// TwinCAT 3 PLC project PLC
// ProgramVersion: 3.1.4022.1
// CompilerDefines: VISU_USEWSTRING
// libraries:
//   Tc2_Drive, * (Beckhoff Automation GmbH)
//   Tc2_EtherCAT, * (Beckhoff Automation GmbH)
//   Tc2_MC2, * (Beckhoff Automation GmbH)
//   Tc2_MC2_Drive, * (Beckhoff Automation GmbH)
//   Tc2_NCI, * (Beckhoff Automation GmbH)
//   Tc2_NcKinematicTransformation, * (Beckhoff Automation GmbH)
//   Tc2_Standard, * (Beckhoff Automation GmbH)
//   Tc2_System, * (Beckhoff Automation GmbH)
//   Tc2_Utilities, * (Beckhoff Automation GmbH)
//   Tc3_McCoordinatedMotion, * (Beckhoff Automation GmbH)
//   Tc3_Module, * (Beckhoff Automation GmbH)
//   VisuDialogs, * (System)
//   VisuElemEventTable,1.0.2.0,System
//   VisuSymbols,newest,System
// project tree:
//   DUTs/ uBYTE_BOOL_MX2.TcDUT, uWORD_BOOL_MX2.TcDUT, E_ColumState.TcDUT, E_LineMachineCommand.TcDUT, E_LineMachineMode.TcDUT, E_MachineCommand.TcDUT, E_MachineMode.TcDUT, E_MachineState.TcDUT, ST_AX5000Diag.TcDUT, ST_ChannelSignals.TcDUT
//   DUTs/E_CaseCloser/ E_CaseCloserMachineState.TcDUT
//   DUTs/E_CaseErector/ E_CaseErectorMachineState.TcDUT
//   DUTs/E_Gantry/ E_GantryMachineState.TcDUT
//   DUTs/HMI/ ST_MachineMode.TcDUT, ST_ManualMode.TcDUT
//   DUTs/NCI/ E_NCIOpModes.TcDUT, ST_NCIChannelState.TcDUT
//   GVLs/ Global_HMI.TcGVL, GVL.TcGVL, GVL_AXIS.TcGVL, GVL_EventsSimple.TcGVL, GVL_GLOBAL.TcGVL, GVL_HMI.TcGVL, GVL_IO.TcGVL, GVL_IO_K.TcGVL, GVL_IO_P.TcGVL, GVL_Kolumna.TcGVL, GVL_Machine.TcGVL, GVL_MachineMaintenance.TcGVL, GVL_NCI.TcGVL, GVL_Omron.TcGVL, GVL_Recipe.TcGVL, GVL_RecipeTable.TcGVL, GVL_SafetyFrom_RT2.TcGVL, GVL_Zak_IO.TcGVL
//   / PlcTask.TcTTO, Recepty.TcTTO, VISU_TASK.TcTTO
//   POUs/Eventy/ FB_SimpleEventLog.TcPOU, P_EventsSimple.TcPOU
//   POUs/FB/ FB_AxisDiag.TcPOU, FB_Button.TcPOU, FB_INV000_MX2_Alarm.TcPOU, FB_INV003_MX2_ECT.TcPOU, FB_Kierownica.TcPOU, FB_K_Auto.TcPOU, FB_Licznik.TcPOU, FB_Magazyn.TcPOU, FB_MX2.TcPOU, FB_MX2_POS.TcPOU, FB_Prawidlo.TcPOU, F_4BYTES_TO_DWORD.TcPOU
//   POUs/Programy/Hbot/AxisOnline/DUTsAxisOnline/FBsIO/ ST_FBCoESetPositionOffsetIO.TcDUT, ST_FBGetDriveRefIO.TcDUT, ST_FBHoldingBrakeCtrlIO.TcDUT, ST_FBMotorMonitoringIO.TcDUT, ST_FBNcSWLimitSwitchCtrlIO.TcDUT, ST_FBReadChannelErrorCodeIO.TcDUT, ST_FBSetPositionOffsetIO.TcDUT, ST_McAxisOnlineErrorCollection.TcDUT, ST_McAxisStatus.TcDUT, ST_MCHaltIO.TcDUT, ST_MCHomeIO.TcDUT, ST_MCJogIO.TcDUT, ST_MCMoveAbsoluteIO.TcDUT, ST_MCMoveModuloIO.TcDUT, ST_MCMoveRelativeIO.TcDUT, ST_MCMoveVelocityIO.TcDUT, ST_MCPowerIO.TcDUT, ST_MCReadDriveAddressIO.TcDUT, ST_MCReadParameterSetIO.TcDUT, ST_MCResetIO.TcDUT, ST_MCSetPositionIO.TcDUT, ST_MCStopIO.TcDUT
//   POUs/Programy/Hbot/AxisOnline/DUTsAxisOnline/ ST_AX5000Diag_1.TcDUT, ST_McAxisOnline.TcDUT
//   POUs/Programy/Hbot/AxisOnline/POUsAxisOnline/AX5000/ FB_AxisDiag_1.TcPOU, FB_ChangeEtherCATSlaveState.TcPOU, FB_HoldingBrakeCtrlAX5000.TcPOU, FB_McAxisOnlineAX5000.TcPOU, FB_MotorMonitoringAX5000.TcPOU, FB_SetPositionOffset.TcPOU
//   POUs/Programy/Hbot/AxisOnline/POUsAxisOnline/FBs/ FB_FilterEx.TcPOU, FB_GetDriveRef.TcPOU, FB_NcSWLimitSwitchCtrl.TcPOU
//   POUs/Programy/Hbot/NCI/1_CTRL/ FB_ConfirmMFunc.TcPOU, FB_EStop.TcPOU, FB_LoadStart.TcPOU, FB_SetOpModeSingleStep.TcPOU, FB_StepOnAfterEStop.TcPOU, F_SetOverride.TcPOU
//   POUs/Programy/Hbot/NCI/2_GROUPS/ FB_BuildGroup.TcPOU, FB_NCIChannel.TcPOU, FB_ReleaseAllGroups.TcPOU, FB_ReleaseGroup.TcPOU, PRG_GroupAxesToNCI.TcPOU
//   POUs/Programy/Hbot/NCI/3_OPMODES/ FB_NCIAutomatic.TcPOU, FB_NCI_MDI.TcPOU
//   POUs/Programy/Hbot/NCI/9_MISC/ FB_ReadRParams.TcPOU, FB_WriteRParams.TcPOU, PRG_GetFastMFunctions.TcPOU
//   POUs/Programy/Hbot/NCI/ PRG_ChannelHandler.TcPOU
//   POUs/Programy/Hbot/NCI/Util/ FB_Blinker.TcPOU
//   POUs/Programy/Hbot/ PRG_KinTrans.TcPOU, P_Hbot_V3.TcPOU, P_ModeStateManager.TcPOU
//   POUs/Programy/ MAIN.TcPOU, PRG_CaseErector.TcPOU, PRG_Kartoniarka.TcPOU, PRG_Kierownica.TcPOU, PRG_CaseMachineMode.TcPOU, PRG_Zaklejarka.TcPOU
//   POUs/RecipeManager/ RecipeManagement.TcPOU
//   VISUs/ GlobalTextList.TcGTLO, Glowna.TcVIS, HMI.TcVIS, IP_Obrazki.TcIPO (not stored), Alarmy.TcVIS, Kartoniarka.TcVIS, Keypad.TcVIS, Kierwonica.TcVIS, mssgbox.TcVIS, PH_AxisOnline.TcVIS, PH_AxisOnline_1.TcVIS, PH_Motor.TcVIS, PH_NcAxis.TcVIS, Ploter.TcVIS, Statystyki.TcVIS, RecipeManager.TcRMO (not stored), Serwis.TcVIS, Visualization.TcVIS, VisualizationManager.TcVMO (not stored), Zaklejarka.TcVIS
// real-time tasks:
//   TASK PlcTask: cycle T#10ms, priority 20, ADS port 350
//   TASK VISU_TASK: cycle T#100000us, priority 30, ADS port 351
//   TASK SafetyTask: cycle T#10ms, priority 21, ADS port 352
//   TASK Recepty: cycle T#50000us, priority 1, ADS port 353
// motion (NC):
//   TASK NC-Task 1 SAF: cycle T#2ms, priority 4, ADS port 501
//   TASK NC-Task 1 SVB: cycle T#10ms, priority 8, ADS port 511
//   AXIS Axis 1 S_Kartoniarka (id 1)
//     Dynamic: Jerk=2249.99
//     Velo: Maximum=3000
//     OtherSettings: AllowMotionCmdToSlave=true
//     encoder EncType=19
//       EncPara: ScaleFactorNumerator=2.16e-06, MaxCount=#xffffffff, ReferenceSystem=1
//     drive DrvType=16
//       DrvPara: MaxCount=#xffffffff, DriveControlDWord=#x00000100
//         Analog: VeloReferenz=3100, ScaleFactorActTorque=0.1
//         TimeComp: TaskDelayCycles=1
//     controller CtrType=1
//       CtrPara: PriorControlFactor=1
//         Observer: BandWidth=20
//   AXIS Axis 2 S_Kierownica (id 2)
//     OtherSettings: AllowMotionCmdToSlave=true
//     encoder EncType=19
//       EncPara: ScaleFactorNumerator=2.16e-06, MaxCount=#xffffffff, ReferenceSystem=1
//     drive DrvType=16
//       DrvPara: MaxCount=#xffffffff, DriveControlDWord=#x00000100
//         Analog: ScaleFactorActTorque=0.1
//         TimeComp: TaskDelayCycles=1
//     controller CtrType=1
//       CtrPara: PriorControlFactor=1
//         Observer: BandWidth=20
//   AXIS Axis 3 Enc (id 3)
//     OtherSettings: AllowMotionCmdToSlave=true
//     encoder EncType=4
//       EncPara: ScaleFactorNumerator=0.0004, ModuloFactor=2000, MaxCount=#x0000ffff
//     drive DrvType=5
//       Analog: ScaleFactorActTorque=0.1
//       TimeComp: TaskDelayCycles=1
//     controller CtrType=1
//       CtrPara: PriorControlFactor=1
//         Observer: BandWidth=20
//   AXIS MC_MFalownik (id 4)
//     OtherSettings: AllowMotionCmdToSlave=true
//     encoder EncType=1
//     drive DrvType=5
//       Analog: ScaleFactorActTorque=0.1
//       TimeComp: TaskDelayCycles=1
//     controller CtrType=1
//       CtrPara: PriorControlFactor=1
//         Observer: BandWidth=20
//   AXIS Mcs_X_Virtual (id 5)
//     Dynamic: Acceleration=2300, Deceleration=2300, Jerk=28000
//     Velo: SlowManual=20, FastManual=100, Maximum=1000
//     OtherSettings: AllowMotionCmdToSlave=true
//     encoder EncType=1
//       SoftEndMinControl: Enable=true
//       SoftEndMaxControl: Enable=true, Range=1152
//     drive DrvType=5
//       Analog: VeloReferenz=1200, ScaleFactorActTorque=0.1
//       TimeComp: TaskDelayCycles=1
//     controller CtrType=1
//       CtrPara: PriorControlFactor=1
//         Observer: BandWidth=20
//   AXIS Mcs_Y_Virtual (id 6)
//     Dynamic: Acceleration=2300, Deceleration=2300, Jerk=28000
//     Velo: SlowManual=20, FastManual=100, Maximum=1000
//     OtherSettings: AllowMotionCmdToSlave=true
//     encoder EncType=1
//       SoftEndMinControl: Enable=true
//       SoftEndMaxControl: Enable=true, Range=735
//     drive DrvType=5
//       Analog: VeloReferenz=1200, ScaleFactorActTorque=0.1
//       TimeComp: TaskDelayCycles=1
//     controller CtrType=1
//       CtrPara: PriorControlFactor=1
//         Observer: BandWidth=20
//   AXIS Acs_X_hw (id 7)
//     Dynamic: Acceleration=4000, Deceleration=4000, Jerk=120000
//     Velo: RefSearch=10.3207170410156, RefSync=10.3207170410156, SlowManual=51.6035852050781, FastManual=309.621511230469, Fast=1032.07170410156, Maximum=1032.07
//     OtherSettings: AllowMotionCmdToSlave=true
//     encoder EncType=8
//       EncPara: ScaleFactorNumerator=18, ScaleFactorDenominator=1048576, Inverse=true, EncMode=3, MaxCount=#xffffffff
//     drive DrvType=9
//       DrvPara: Inverse=true, MaxCount=#xffffffff, DriveControlDWord=#x00030100
//         Analog: VeloReferenz=1135.27887451172, VeloScale=1.02400649589962, ScaleFactorActTorque=0.1
//         TimeComp: TaskDelayCycles=1
//     controller CtrType=1
//       CtrPara: PriorControlFactor=1
//         Observer: BandWidth=20
//   AXIS Acs_Y_Hw (id 8)
//     Dynamic: Acceleration=4000, Deceleration=4000, Jerk=120000
//     Velo: RefSearch=10.3207170410156, RefSync=10.3207170410156, SlowManual=51.6035852050781, FastManual=309.621511230469, Fast=1032.07170410156, Maximum=1032.07
//     OtherSettings: AllowMotionCmdToSlave=true
//     encoder EncType=8
//       EncPara: ScaleFactorNumerator=18, ScaleFactorDenominator=1048576, Inverse=true, EncMode=3, MaxCount=#xffffffff
//     drive DrvType=9
//       DrvPara: Inverse=true, MaxCount=#xffffffff, DriveControlDWord=#x00030100
//         Analog: VeloReferenz=1135.27887451172, VeloScale=1.02400649589962, ScaleFactorActTorque=0.1
//         TimeComp: TaskDelayCycles=1
//     controller CtrType=1
//       CtrPara: PriorControlFactor=1
//         Observer: BandWidth=20
// I/O:
//   DEVICE Device 3 (EtherCAT), AmsNetId 169.254.71.253.4.1
//     Term 1 (EK1100) [EK1100 EtherCAT Coupler (2A E-Bus)]
//       Term 2 (EL6910) [EL6910, TwinSAFE PLC]
//       Term 3 (EL1904) [EL1904, 4 Ch. Safety Input 24V, TwinSAFE]
//         modules: Module 1 (FSOES)
//       Term 4 (EL1904) [EL1904, 4 Ch. Safety Input 24V, TwinSAFE]
//         modules: Module 1 (FSOES)
//       Term 5 (EL2904) [EL2904, 4 Ch. Safety Output 24V, 0.5A, TwinSAFE]
//         modules: Module 1 (FSOES), Module 2 (DO)
//       Term 6 (EL1008) [EL1008 8Ch. Dig. Input 24V, 3ms]
//       Term 7 (EL2008) [EL2008 8Ch. Dig. Output 24V, 0.5A]
//       Term 21 (EL1008) [EL1008 8Ch. Dig. Input 24V, 3ms]
//       Term 9 (EL9011) [EL9011 End Terminal]
//     Drive 10 (R88D-1SN04H-ECT) [R88D-1SN04H-ECT 200V/400W ServoDrive]
//       modules: Module 1 (Safety Process Data)
//     Box 11 (3G3AX-MX2-ECT) [3G3AX-MX2-ECT EtherCAT Communication Unit for 3G3MX2]
//     Box 12 (3G3AX-MX2-ECT) [3G3AX-MX2-ECT EtherCAT Communication Unit for 3G3MX2]
//     Box 13 (BNI ECT-507-005-Z040) [BNI ECT-507-005-Z040 (BNI009U)]
//       modules: Module 1 (IOL_I/O_8/_2byte), Module 2 (IOL_O_2byte), Module 3 (IOL_I/O_8/_2byte), Module 4 (STD_IN_1bit), Module 33 (OUTPUT_PIN2_4CH)
//     Term 14 (EK1100) [EK1100 EtherCAT Coupler (2A E-Bus)]
//       Term 15 (EL1008) [EL1008 8Ch. Dig. Input 24V, 3ms]
//       Term 16 (EL2008) [EL2008 8Ch. Dig. Output 24V, 0.5A]
//       Term 17 (EL1904) [EL1904, 4 Ch. Safety Input 24V, TwinSAFE]
//         modules: Module 1 (FSOES)
//       Term 18 (EL1904) [EL1904, 4 Ch. Safety Input 24V, TwinSAFE]
//         modules: Module 1 (FSOES)
//       Term 19 (EL2904) [EL2904, 4 Ch. Safety Output 24V, 0.5A, TwinSAFE]
//         modules: Module 1 (FSOES), Module 2 (DO)
//       Term 32 (EL2904) [EL2904, 4 Ch. Safety Output 24V, 0.5A, TwinSAFE]
//         modules: Module 1 (FSOES), Module 2 (DO)
//       Term 20 (EL9011) [EL9011 End Terminal]
//     Box 21 (3G3AX-MX2-ECT) [3G3AX-MX2-ECT EtherCAT Communication Unit for 3G3MX2]
//     Drive 22 (R88D-1SN04H-ECT) [R88D-1SN04H-ECT 200V/400W ServoDrive]
//       modules: Module 1 (Safety Process Data)
//     Term 23 (EK1100) [EK1100 EtherCAT Coupler (2A E-Bus)]
//       Term 24 (EL1904) [EL1904, 4 Ch. Safety Input 24V, TwinSAFE]
//         modules: Module 1 (FSOES)
//       Term 25 (EL1904) [EL1904, 4 Ch. Safety Input 24V, TwinSAFE]
//         modules: Module 1 (FSOES)
//       Term 26 (EL2904) [EL2904, 4 Ch. Safety Output 24V, 0.5A, TwinSAFE]
//         modules: Module 1 (FSOES), Module 2 (DO)
//       Term 27 (EL2904) [EL2904, 4 Ch. Safety Output 24V, 0.5A, TwinSAFE]
//         modules: Module 1 (FSOES), Module 2 (DO)
//       Term 28 (EL1008) [EL1008 8Ch. Dig. Input 24V, 3ms]
//       Term 29 (EL2008) [EL2008 8Ch. Dig. Output 24V, 0.5A]
//       Term 30 (EK1122) [EK1122 2 port EtherCAT junction]
//       Term 31 (EL9011) [EL9011 End Terminal]
//     Box 32 (3G3AX-MX2-ECT) [3G3AX-MX2-ECT EtherCAT Communication Unit for 3G3MX2]
//     Drive 33 (AX5203-0000-0203) [AX5203-0000-0203 EtherCAT Drive (SoE, 2 Ch.)]
//     Term 34 (EK1100) [EK1100 EtherCAT Coupler (2A E-Bus)]
//       Term 35 (EL6070) [EL6070 1Ch. Licensing-Terminal]
//       Term 36 (EL1008) [EL1008 8Ch. Dig. Input 24V, 3ms]
//       Term 37 (EL2008) [EL2008 8Ch. Dig. Output 24V, 0.5A]
//       Term 38 (EL1904) [EL1904, 4 Ch. Safety Input 24V, TwinSAFE]
//         modules: Module 1 (FSOES)
//       Term 39 (EL1904) [EL1904, 4 Ch. Safety Input 24V, TwinSAFE]
//         modules: Module 1 (FSOES)
//       Term 40 (EL2904) [EL2904, 4 Ch. Safety Output 24V, 0.5A, TwinSAFE]
//         modules: Module 1 (FSOES), Module 2 (DO)
//       Term 41 (EL9011) [EL9011 End Terminal]
//     Box 42 (3G3AX-MX2-ECT) [3G3AX-MX2-ECT EtherCAT Communication Unit for 3G3MX2]
// variable links:
//   Device 3 (EtherCAT) <-> Device 3 (EtherCAT)/Term 1 (EK1100)/Term 2 (EL6910)
//     Term 1 (EK1100)/Term 3 (EL1904)/Module 1 (FSOES)/TxPDO/FSOE <-> ConnectionOutputs/Message_63 RxPDO
//     Term 14 (EK1100)/Term 17 (EL1904)/Module 1 (FSOES)/TxPDO/FSOE <-> ConnectionOutputs/Message_69 RxPDO
//     Term 23 (EK1100)/Term 27 (EL2904)/Module 1 (FSOES)/TxPDO/FSOE <-> ConnectionOutputs/Message_59 RxPDO
//     Term 34 (EK1100)/Term 38 (EL1904)/Module 1 (FSOES)/TxPDO/FSOE <-> ConnectionOutputs/Message_67 RxPDO
//     Term 34 (EK1100)/Term 40 (EL2904)/Module 1 (FSOES)/TxPDO/FSOE <-> ConnectionOutputs/Message_66 RxPDO
//     Term 14 (EK1100)/Term 19 (EL2904)/Module 1 (FSOES)/RxPDO/FSOE <-> ConnectionInputs/Message_65 TxPDO
//   Device 3 (EtherCAT) <-> Device 3 (EtherCAT)/Term 1 (EK1100)/Term 3 (EL1904)
//     Term 1 (EK1100)/Term 2 (EL6910)/ConnectionInputs/Message_63 TxPDO <-> Module 1 (FSOES)/RxPDO/FSOE
//   Device 3 (EtherCAT) <-> Device 3 (EtherCAT)/Term 1 (EK1100)/Term 4 (EL1904)
//     Term 1 (EK1100)/Term 2 (EL6910)/ConnectionInputs/Message_64 TxPDO <-> Module 1 (FSOES)/RxPDO/FSOE
//     Term 1 (EK1100)/Term 2 (EL6910)/ConnectionOutputs/Message_64 RxPDO <-> Module 1 (FSOES)/TxPDO/FSOE
//   Device 3 (EtherCAT) <-> Device 3 (EtherCAT)/Term 1 (EK1100)/Term 5 (EL2904)
//     Term 1 (EK1100)/Term 2 (EL6910)/ConnectionInputs/Message_52 TxPDO <-> Module 1 (FSOES)/RxPDO/FSOE
//     Term 1 (EK1100)/Term 2 (EL6910)/ConnectionOutputs/Message_52 RxPDO <-> Module 1 (FSOES)/TxPDO/FSOE
//   Device 3 (EtherCAT) <-> Device 3 (EtherCAT)/Term 14 (EK1100)/Term 17 (EL1904)
//     Term 1 (EK1100)/Term 2 (EL6910)/ConnectionInputs/Message_69 TxPDO <-> Module 1 (FSOES)/RxPDO/FSOE
//   Device 3 (EtherCAT) <-> Device 3 (EtherCAT)/Term 14 (EK1100)/Term 19 (EL2904)
//     Term 1 (EK1100)/Term 2 (EL6910)/ConnectionOutputs/Message_65 RxPDO <-> Module 1 (FSOES)/TxPDO/FSOE
//   Device 3 (EtherCAT) <-> Device 3 (EtherCAT)/Term 23 (EK1100)/Term 24 (EL1904)
//     Term 1 (EK1100)/Term 2 (EL6910)/ConnectionInputs/Message_68 TxPDO <-> Module 1 (FSOES)/RxPDO/FSOE
//     Term 1 (EK1100)/Term 2 (EL6910)/ConnectionOutputs/Message_68 RxPDO <-> Module 1 (FSOES)/TxPDO/FSOE
//   Device 3 (EtherCAT) <-> Device 3 (EtherCAT)/Term 23 (EK1100)/Term 27 (EL2904)
//     Term 1 (EK1100)/Term 2 (EL6910)/ConnectionInputs/Message_59 TxPDO <-> Module 1 (FSOES)/RxPDO/FSOE
//   Device 3 (EtherCAT) <-> Device 3 (EtherCAT)/Term 34 (EK1100)/Term 38 (EL1904)
//     Term 1 (EK1100)/Term 2 (EL6910)/ConnectionInputs/Message_67 TxPDO <-> Module 1 (FSOES)/RxPDO/FSOE
//   Device 3 (EtherCAT) <-> Device 3 (EtherCAT)/Term 34 (EK1100)/Term 40 (EL2904)
//     Term 1 (EK1100)/Term 2 (EL6910)/ConnectionInputs/Message_66 TxPDO <-> Module 1 (FSOES)/RxPDO/FSOE
//   NC-Task 1 SAF/Axes/Acs_X_hw <-> Device 3 (EtherCAT)/Drive 33 (AX5203-0000-0203)
//     Drive/Inputs/In/nDataIn1 <-> AT 1/Following distance
//     Drive/Inputs/In/nDataIn3[0] <-> AT 1/Torque feedback value
//     Drive/Inputs/In/nDcOutputTime <-> InfoData/DcOutputShift
//     Drive/Inputs/In/nState1 <-> AT 1/Drive status word @bit 8
//     Drive/Inputs/In/nState2 <-> AT 1/Drive status word
//     Drive/Inputs/In/nState4 @bit 1 <-> WcState/InputToggle
//     Drive/Inputs/In/nState4 <-> WcState/WcState
//     Drive/Outputs/Out/nCtrl1 <-> MDT 1/Master control word @bit 8
//     Drive/Outputs/Out/nDataOut1 <-> MDT 1/Position command value
//     Enc/Inputs/In/nDataIn1 <-> AT 1/Position feedback 1 value
//     Enc/Inputs/In/nDcInputTime <-> InfoData/DcInputShift
//     Enc/Inputs/In/nState4 @bit 1 <-> WcState/InputToggle
//     Enc/Inputs/In/nState4 <-> WcState/WcState
//   NC-Task 1 SAF/Axes/Acs_Y_Hw <-> Device 3 (EtherCAT)/Drive 33 (AX5203-0000-0203)
//     Drive/Inputs/In/nDataIn1 <-> AT 2/Following distance
//     Drive/Inputs/In/nDataIn3[0] <-> AT 2/Torque feedback value
//     Drive/Inputs/In/nDcOutputTime <-> InfoData/DcOutputShift
//     Drive/Inputs/In/nState1 <-> AT 2/Drive status word @bit 8
//     Drive/Inputs/In/nState2 <-> AT 2/Drive status word
//     Drive/Inputs/In/nState4 @bit 1 <-> WcState/InputToggle
//     Drive/Inputs/In/nState4 <-> WcState/WcState
//     Drive/Outputs/Out/nCtrl1 <-> MDT 2/Master control word @bit 8
//     Drive/Outputs/Out/nDataOut1 <-> MDT 2/Position command value
//     Enc/Inputs/In/nDataIn1 <-> AT 2/Position feedback 1 value
//     Enc/Inputs/In/nDcInputTime <-> InfoData/DcInputShift
//     Enc/Inputs/In/nState4 @bit 1 <-> WcState/InputToggle
//     Enc/Inputs/In/nState4 <-> WcState/WcState
//   NC-Task 1 SAF/Axes/Axis 1 S_Kartoniarka <-> Device 3 (EtherCAT)/Drive 10 (R88D-1SN04H-ECT)
//     Drive/Inputs/In/nDataIn1 <-> 258th transmit PDO Mapping/Following error actual value
//     Drive/Inputs/In/nDataIn3[0] <-> 258th transmit PDO Mapping/Torque actual value
//     Drive/Inputs/In/nDcOutputTime <-> InfoData/DcOutputShift
//     Drive/Inputs/In/nState1 <-> 258th transmit PDO Mapping/Statusword
//     Drive/Inputs/In/nState2 <-> 258th transmit PDO Mapping/Statusword @bit 8
//     Drive/Inputs/In/nState4 @bit 1 <-> WcState/InputToggle
//     Drive/Inputs/In/nState4 <-> WcState/WcState
//     Drive/Outputs/Out/nCtrl1 <-> 258th receive PDO Mapping/Controlword
//     Drive/Outputs/Out/nCtrl2 <-> 258th receive PDO Mapping/Controlword @bit 8
//     Drive/Outputs/Out/nDataOut1 <-> 258th receive PDO Mapping/Target position
//     Enc/Inputs/In/nDataIn1 <-> 258th transmit PDO Mapping/Position actual value
//     Enc/Inputs/In/nDataIn3 <-> 258th transmit PDO Mapping/Touch probe pos1 pos value
//     Enc/Inputs/In/nDataIn5 <-> 258th transmit PDO Mapping/Touch probe pos2 pos value
//     Enc/Inputs/In/nDcInputTime <-> InfoData/DcInputShift
//     Enc/Inputs/In/nState4 @bit 1 <-> WcState/InputToggle
//     Enc/Inputs/In/nState4 <-> WcState/WcState
//     Enc/Inputs/In/nState5 <-> 258th transmit PDO Mapping/Touch probe status
//     Enc/Inputs/In/nState6 <-> 258th transmit PDO Mapping/Touch probe status @bit 8
//     Enc/Outputs/Out/nCtrl5 <-> 258th receive PDO Mapping/Touch probe function
//     Enc/Outputs/Out/nCtrl6 <-> 258th receive PDO Mapping/Touch probe function @bit 8
//   NC-Task 1 SAF/Axes/Axis 2 S_Kierownica <-> Device 3 (EtherCAT)/Drive 22 (R88D-1SN04H-ECT)
//     Drive/Inputs/In/nDataIn1 <-> 258th transmit PDO Mapping/Following error actual value
//     Drive/Inputs/In/nDataIn3[0] <-> 258th transmit PDO Mapping/Torque actual value
//     Drive/Inputs/In/nDcOutputTime <-> InfoData/DcOutputShift
//     Drive/Inputs/In/nState1 <-> 258th transmit PDO Mapping/Statusword
//     Drive/Inputs/In/nState2 <-> 258th transmit PDO Mapping/Statusword @bit 8
//     Drive/Inputs/In/nState4 @bit 1 <-> WcState/InputToggle
//     Drive/Inputs/In/nState4 <-> WcState/WcState
//     Drive/Outputs/Out/nCtrl1 <-> 258th receive PDO Mapping/Controlword
//     Drive/Outputs/Out/nCtrl2 <-> 258th receive PDO Mapping/Controlword @bit 8
//     Drive/Outputs/Out/nDataOut1 <-> 258th receive PDO Mapping/Target position
//     Enc/Inputs/In/nDataIn1 <-> 258th transmit PDO Mapping/Position actual value
//     Enc/Inputs/In/nDataIn3 <-> 258th transmit PDO Mapping/Touch probe pos1 pos value
//     Enc/Inputs/In/nDataIn5 <-> 258th transmit PDO Mapping/Touch probe pos2 pos value
//     Enc/Inputs/In/nDcInputTime <-> InfoData/DcInputShift
//     Enc/Inputs/In/nState4 @bit 1 <-> WcState/InputToggle
//     Enc/Inputs/In/nState4 <-> WcState/WcState
//     Enc/Inputs/In/nState5 <-> 258th transmit PDO Mapping/Touch probe status
//     Enc/Inputs/In/nState6 <-> 258th transmit PDO Mapping/Touch probe status @bit 8
//     Enc/Outputs/Out/nCtrl5 <-> 258th receive PDO Mapping/Touch probe function
//     Enc/Outputs/Out/nCtrl6 <-> 258th receive PDO Mapping/Touch probe function @bit 8
//   PLC/PLC Instance <-> Device 3 (EtherCAT)/Box 11 (3G3AX-MX2-ECT)
//     PlcTask Inputs/GVL_Omron.iOmronErectorAcc <-> 1st transmit PDO Mapping/F002 1st Acceleration Time 1
//     PlcTask Inputs/GVL_Omron.iOmronErectorDcc <-> 2nd transmit PDO Mapping/F003 1st Deceleration Time 1
//     PlcTask Inputs/GVL_Omron.iOmron_1_ActVelo <-> 258th transmit PDO Mapping/Output frequency monitor
//     PlcTask Inputs/GVL_Omron.wOmron_1_Status <-> 258th transmit PDO Mapping/Status
//     PlcTask Outputs/GVL_Omron.iOmron_1_SeVelo <-> 258th receive PDO Mapping/Frequency reference
//     PlcTask Outputs/GVL_Omron.wOmron_1_Control <-> 258th receive PDO Mapping/Command
//   PLC/PLC Instance <-> Device 3 (EtherCAT)/Box 13 (BNI ECT-507-005-Z040)
//     PlcTask Inputs/GVL_IO.Kl_1_cof <-> Module 3 (IOL_I/O_8/_2byte)/TxPDO/input byte 0[5]
//     PlcTask Inputs/GVL_IO.Kl_2_cof <-> Module 3 (IOL_I/O_8/_2byte)/TxPDO/input byte 0[6]
//     PlcTask Inputs/GVL_IO.Kl_1_wyp <-> Module 3 (IOL_I/O_8/_2byte)/TxPDO/input byte 1[5]
//     PlcTask Inputs/GVL_IO.Kl_2_wyp <-> Module 3 (IOL_I/O_8/_2byte)/TxPDO/input byte 0[4]
//     PlcTask Inputs/GVL_IO.Skos_cof <-> Module 3 (IOL_I/O_8/_2byte)/TxPDO/input byte 0[3]
//     PlcTask Inputs/GVL_IO.Skos_wyp <-> Module 3 (IOL_I/O_8/_2byte)/TxPDO/input byte 0[2]
//     PlcTask Inputs/GVL_IO.Wyp_cof <-> Module 3 (IOL_I/O_8/_2byte)/TxPDO/input byte 0[1]
//     PlcTask Inputs/GVL_IO.Wyp_wys <-> Module 3 (IOL_I/O_8/_2byte)/TxPDO/input byte 0[0]
//     PlcTask Inputs/GVL_IO.Zeb_Cof <-> Module 3 (IOL_I/O_8/_2byte)/TxPDO/input byte 1[7]
//     PlcTask Inputs/GVL_IO.Zeb_Wyp <-> Module 3 (IOL_I/O_8/_2byte)/TxPDO/input byte 0[7]
//     PlcTask Outputs/GVL_IO.IOLinkCh1T <-> Module 33 (OUTPUT_PIN2_4CH)/IO Output Pin 2 (4 Ch)/Output Pin 2 of Ch1
//     PlcTask Outputs/GVL_IO.P_Vac <-> Module 1 (IOL_I/O_8/_2byte)/RxPDO/output byte 0[3]
//     PlcTask Outputs/GVL_IO.S_Kl_1 <-> Module 1 (IOL_I/O_8/_2byte)/RxPDO/output byte 0[1]
//     PlcTask Outputs/GVL_IO.S_Kl_2 <-> Module 1 (IOL_I/O_8/_2byte)/RxPDO/output byte 0[5]
//     PlcTask Outputs/GVL_IO.S_Wypych <-> Module 1 (IOL_I/O_8/_2byte)/RxPDO/output byte 0[6]
//     PlcTask Outputs/GVL_IO.S_Zeb <-> Module 1 (IOL_I/O_8/_2byte)/RxPDO/output byte 0[0]
//     PlcTask Outputs/GVL_IO.S_skos <-> Module 1 (IOL_I/O_8/_2byte)/RxPDO/output byte 0[4]
//     PlcTask Outputs/GVL_Kolumna.Segment_1 <-> Module 2 (IOL_O_2byte)/RxPDO/output byte 0
//     PlcTask Outputs/GVL_Kolumna.Segment_2 <-> Module 2 (IOL_O_2byte)/RxPDO/output byte 1
//   PLC/PLC Instance <-> Device 3 (EtherCAT)/Box 21 (3G3AX-MX2-ECT)
//     PlcTask Inputs/GVL_Omron.iOmron_Kier_ActVelo <-> 258th transmit PDO Mapping/Output frequency monitor
//     PlcTask Inputs/GVL_Omron.wOmron_Kier_Status <-> 258th transmit PDO Mapping/Status
//     PlcTask Outputs/GVL_Omron.iOmron_Kier_SeVelo <-> 258th receive PDO Mapping/Frequency reference
//     PlcTask Outputs/GVL_Omron.wOmron_Kier_Control <-> 258th receive PDO Mapping/Command
//   PLC/PLC Instance <-> Device 3 (EtherCAT)/Box 32 (3G3AX-MX2-ECT)
//     PlcTask Inputs/GVL_Omron.iOmron_Pl_ActVelo <-> 258th transmit PDO Mapping/Output frequency monitor
//     PlcTask Inputs/GVL_Omron.wOmron_Pl_Status <-> 258th transmit PDO Mapping/Status
//     PlcTask Outputs/GVL_Omron.iOmron_Pl_SeVelo <-> 258th receive PDO Mapping/Frequency reference
//     PlcTask Outputs/GVL_Omron.wOmron_Pl_Control <-> 258th receive PDO Mapping/Command
//   PLC/PLC Instance <-> Device 3 (EtherCAT)/Box 42 (3G3AX-MX2-ECT)
//     PlcTask Inputs/GVL_Omron.iOmron_Za_ActVelo <-> 258th transmit PDO Mapping/Output frequency monitor
//     PlcTask Inputs/GVL_Omron.wOmron_Za_Status <-> 258th transmit PDO Mapping/Status
//     PlcTask Outputs/GVL_Omron.iOmron_Za_SeVelo <-> 258th receive PDO Mapping/Frequency reference
//     PlcTask Outputs/GVL_Omron.wOmron_Za_Control <-> 258th receive PDO Mapping/Command
//   PLC/PLC Instance <-> Device 3 (EtherCAT)/Term 1 (EK1100)/Term 21 (EL1008)
//     PlcTask Inputs/GVL_IO.bCzujnik_Trzymacz1 <-> Channel 7/Input
//   PLC/PLC Instance <-> Device 3 (EtherCAT)/Term 1 (EK1100)/Term 6 (EL1008)
//     PlcTask Inputs/GVL_IO.b1K{1..8} <-> Channel {1..8}/Input  (8 links)
//   PLC/PLC Instance <-> Device 3 (EtherCAT)/Term 1 (EK1100)/Term 7 (EL2008)
//     PlcTask Outputs/GVL_IO.K1K{1..8} <-> Channel {1..8}/Output  (8 links)
//   PLC/PLC Instance <-> Device 3 (EtherCAT)/Term 14 (EK1100)/Term 15 (EL1008)
//     PlcTask Inputs/GVL_IO_K.b4B{1..8} <-> Channel {1..8}/Input  (8 links)
//   PLC/PLC Instance <-> Device 3 (EtherCAT)/Term 14 (EK1100)/Term 16 (EL2008)
//     PlcTask Outputs/GVL_IO_K.bK{1..8} <-> Channel {1..8}/Output  (8 links)
//   PLC/PLC Instance <-> Device 3 (EtherCAT)/Term 23 (EK1100)/Term 28 (EL1008)
//     PlcTask Inputs/GVL_IO_P.b{1..8}B1 <-> Channel {1..8}/Input  (8 links)
//   PLC/PLC Instance <-> Device 3 (EtherCAT)/Term 23 (EK1100)/Term 29 (EL2008)
//     PlcTask Outputs/GVL_IO_P.b{1..8}K1 <-> Channel {1..8}/Output  (8 links)
//   PLC/PLC Instance <-> Device 3 (EtherCAT)/Term 34 (EK1100)/Term 36 (EL1008)
//     PlcTask Inputs/GVL_Zak_IO.b{5..8}B1 <-> Channel {5..8}/Input  (4 links)
//     PlcTask Inputs/GVL_Zak_IO.b_Czujnik_Karton <-> Channel 1/Input
//     PlcTask Inputs/GVL_Zak_IO.b_czujnik_OT <-> Channel 2/Input
//     PlcTask Inputs/GVL_Zak_IO.b_kZamykacz1 <-> Channel 3/Input
//     PlcTask Inputs/GVL_Zak_IO.b_kZamykacz2 <-> Channel 4/Input
//   PLC/PLC Instance <-> Device 3 (EtherCAT)/Term 34 (EK1100)/Term 37 (EL2008)
//     PlcTask Outputs/GVL_Zak_IO.bK{3..8} <-> Channel {3..8}/Output  (6 links)
//     PlcTask Outputs/GVL_Zak_IO.b_Sil_Zamkniecie <-> Channel 1/Output
//   PLC/PLC Instance <-> NC-Task 1 SAF/Axes/Acs_X_hw
//     PlcTask Inputs/P_Hbot_V3.Axis_ACS_X.NcToPlc <-> Outputs/ToPlc
//     PlcTask Outputs/P_Hbot_V3.Axis_ACS_X.PlcToNc <-> Inputs/FromPlc
//   PLC/PLC Instance <-> NC-Task 1 SAF/Axes/Acs_Y_Hw
//     PlcTask Inputs/P_Hbot_V3.Axis_ACS_Y.NcToPlc <-> Outputs/ToPlc
//     PlcTask Outputs/P_Hbot_V3.Axis_ACS_Y.PlcToNc <-> Inputs/FromPlc
//   PLC/PLC Instance <-> NC-Task 1 SAF/Axes/Axis 1 S_Kartoniarka
//     PlcTask Inputs/GVL_AXIS.stAxis1.NcToPlc <-> Outputs/ToPlc
//     PlcTask Outputs/GVL_AXIS.stAxis1.PlcToNc <-> Inputs/FromPlc
//   PLC/PLC Instance <-> NC-Task 1 SAF/Axes/Axis 2 S_Kierownica
//     PlcTask Inputs/GVL_AXIS.stAxis2.NcToPlc <-> Outputs/ToPlc
//     PlcTask Outputs/GVL_AXIS.stAxis2.PlcToNc <-> Inputs/FromPlc
//   PLC/PLC Instance <-> NC-Task 1 SAF/Axes/Axis 3 Enc
//     PlcTask Inputs/GVL_AXIS.EC_Magazyn.NcToPlc <-> Outputs/ToPlc
//     PlcTask Outputs/GVL_AXIS.EC_Magazyn.PlcToNc <-> Inputs/FromPlc
//   PLC/PLC Instance <-> NC-Task 1 SAF/Axes/MC_MFalownik
//     PlcTask Inputs/GVL_AXIS.F_Magazyn.NcToPlc <-> Outputs/ToPlc
//     PlcTask Outputs/GVL_AXIS.F_Magazyn.PlcToNc <-> Inputs/FromPlc
//   PLC/PLC Instance <-> NC-Task 1 SAF/Axes/Mcs_X_Virtual
//     PlcTask Inputs/P_Hbot_V3.Axis_MCS_X.NcToPlc <-> Outputs/ToPlc
//     PlcTask Outputs/P_Hbot_V3.Axis_MCS_X.PlcToNc <-> Inputs/FromPlc
//   PLC/PLC Instance <-> NC-Task 1 SAF/Axes/Mcs_Y_Virtual
//     PlcTask Inputs/P_Hbot_V3.Axis_MCS_Y.NcToPlc <-> Outputs/ToPlc
//     PlcTask Outputs/P_Hbot_V3.Axis_MCS_Y.PlcToNc <-> Inputs/FromPlc
//   PLC/PLC Instance <-> NC-Task 1 SAF/Channel 2
//     PlcTask Inputs/GVL_NCI.arrNCToPLC_NCIChannel_REF[1] <-> Outputs/ToPlc
//     PlcTask Outputs/GVL_NCI.arrPLCToNC_NCIChannel_REF[1] <-> Inputs/FromPlc
//   PLC/PLC Instance <-> NC-Task 1 SAF/HBot
//     PlcTask Inputs/PRG_KinTrans.in_stKinToPlc <-> Outputs/ToPlc
//     PlcTask Outputs/PRG_KinTrans.out_stPlcToKin <-> Inputs/FromPlc
//   PLC/PLC Instance <-> SafetyLogic/SafetyLogic Instance
//     PlcTask Inputs/GVL_SafetyFrom_RT2.bSAFETY_Error <-> SafetyTask Outputs/GVL_IO_SAFETY.bSAFETY_Error
//     PlcTask Inputs/GVL_SafetyFrom_RT2.bSAFETY_FalownikKierPermitionOutSS1 <-> SafetyTask Outputs/GVL_IO_SAFETY.bSAFETY_FalownikKierPermitionOutSS1
//     PlcTask Inputs/GVL_SafetyFrom_RT2.bSAFETY_PermissionSS1 <-> SafetyTask Outputs/GVL_IO_SAFETY.bSAFETY_PermissionOutSS1
//     PlcTask Inputs/GVL_SafetyFrom_RT2.bSAFETY_PermissionSS2 <-> SafetyTask Outputs/GVL_IO_SAFETY.bSAFETY_PermissionOutSS2
//     PlcTask Inputs/GVL_SafetyFrom_RT2.bSAFETY_ResetBusy <-> SafetyTask Outputs/GVL_IO_SAFETY.bSAFETY_ResetBusy
//     PlcTask Inputs/GVL_SafetyFrom_RT2.bSAFETY_ServoKierPermitionOutSS1 <-> SafetyTask Outputs/GVL_IO_SAFETY.bSAFETY_ServoKierPermitionOutSS1
//     PlcTask Inputs/GVL_SafetyFrom_RT2.bSAFETY_ZaklejarkaKierPermitionOutSS1 <-> SafetyTask Outputs/GVL_IO_SAFETY.bSAFETY_ZaklejarkaKierPermitionOutSS1
//     PlcTask Inputs/GVL_SafetyFrom_RT2.dwGroupErrors <-> SafetyTask Outputs/GVL_IO_SAFETY.dwGroupErrors
//     PlcTask Outputs/GVL_SafetyFrom_RT2.bSAFETY_ResetCMD <-> SafetyTask Inputs/GVL_IO_SAFETY.bSAFETY_ResetCMD
//   SafetyLogic/SafetyLogic Instance <-> Device 3 (EtherCAT)/Term 1 (EK1100)/Term 2 (EL6910)
//     SafetyTask Inputs/GVL_IO_SAFETY.bCOM_ERR_TSG1 <-> StandardInputs/Standard Out Var 34
//     SafetyTask Inputs/GVL_IO_SAFETY.bCOM_ERR_TSG2 <-> StandardInputs/Standard Out Var 44
//     SafetyTask Inputs/GVL_IO_SAFETY.bFB_ERR_TSG1 <-> StandardInputs/Standard Out Var 31
//     SafetyTask Inputs/GVL_IO_SAFETY.bFB_ERR_TSG2 <-> StandardInputs/Standard Out Var 45
//     SafetyTask Inputs/GVL_IO_SAFETY.bFalownikKierownicaEStop <-> StandardInputs/Standard Out Var 71
//     SafetyTask Inputs/GVL_IO_SAFETY.bOTHER_ERR_TSG1 <-> StandardInputs/Standard Out Var 37
//     SafetyTask Inputs/GVL_IO_SAFETY.bOTHER_ERR_TSG2 <-> StandardInputs/Standard Out Var 46
//     SafetyTask Inputs/GVL_IO_SAFETY.bSafeStopAX5000 <-> StandardInputs/Standard Out Var 56
//     SafetyTask Inputs/GVL_IO_SAFETY.bSafeStopOmron <-> StandardInputs/Standard Out Var 55
//     SafetyTask Inputs/GVL_IO_SAFETY.bServoKierownicaEStop <-> StandardInputs/Standard Out Var 70
//     SafetyTask Inputs/GVL_IO_SAFETY.bZaklejarkaEStop <-> StandardInputs/Standard Out Var 72
//     SafetyTask Outputs/GVL_IO_SAFETY.bERR_ACK_TSG1 <-> StandardOutputs/Standard In Var 28
//     SafetyTask Outputs/GVL_IO_SAFETY.bERR_ACK_TSG2 <-> StandardOutputs/Standard In Var 42
//     SafetyTask Outputs/GVL_IO_SAFETY.bRUN_STOP_TSG1 <-> StandardOutputs/Standard In Var 25
//     SafetyTask Outputs/GVL_IO_SAFETY.bRUN_STOP_TSG2 <-> StandardOutputs/Standard In Var 43
//     SafetyTask Outputs/GVL_IO_SAFETY.bRestartFBs_TSG1 <-> StandardOutputs/Standard In Var 54

CONFIGURATION PLC
    RESOURCE PLC ON TwinCAT3
        TASK PlcTask(INTERVAL := T#10ms, PRIORITY := 20);
        TASK Recepty(INTERVAL := T#50000us, PRIORITY := 1);
        TASK VISU_TASK(INTERVAL := T#100000us, PRIORITY := 30);
        PROGRAM MAIN WITH PlcTask : MAIN;
        PROGRAM RecipeManagement WITH Recepty : RecipeManagement;
        PROGRAM VISU_PRG WITH VISU_TASK : VISU_PRG;
    END_RESOURCE
END_CONFIGURATION

// ---- DUTs/uBYTE_BOOL_MX2.TcDUT
TYPE uBYTE_BOOL_MX2 :
UNION
	bits 			:ARRAY[0..7] OF BOOL;
	value			:BYTE;
END_UNION
END_TYPE

// ---- DUTs/uWORD_BOOL_MX2.TcDUT
TYPE uWORD_BOOL_MX2 :
UNION
	bits 			:ARRAY [0..15] OF BOOL;
	ch 				:WORD;
	
END_UNION
END_TYPE

// ---- DUTs/E_CaseCloser/E_CaseCloserMachineState.TcDUT
{attribute 'strict'}
{attribute 'qualified_only'}
TYPE E_CaseCloserMachineState :
(
	eIdle					:= 0,
	eAborting				:= 10,
	eAborted				:= 20,
	eStopping				:= 30,
	eStopped				:= 40,
	eStarting				:= 50,
	eRunning				:= 60,
	eReseting				:= 70,
	eRestarting				:= 80,
	eError					:= 1000	
);
END_TYPE

// ---- DUTs/E_CaseErector/E_CaseErectorMachineState.TcDUT
{attribute 'strict'}
{attribute 'qualified_only'}
TYPE E_CaseErectorMachineState :
(
	eIdle					:= 0,
	eAborting				:= 10,
	eAborted				:= 20,
	eStopping				:= 30,
	eStopped				:= 40,
	eStarting				:= 50,
	eRunning				:= 60,
	eReseting				:= 70,
	eRestarting				:= 80,
	eError					:= 1000	
);
END_TYPE

// ---- DUTs/E_ColumState.TcDUT
{attribute 'qualified_only'}
{attribute 'strict'}
TYPE E_ColumState :
(	
	eIdle			:=0,
	eClear_Estop	:=10,
	eSafety_Ready	:=20,
	eReadyToWork	:=30,
	eRun			:=40,
	eError			:=50,
	eEstopPush		:=60,	
	eManualMode		:=70,
	eWork		:=80
);
END_TYPE

// ---- DUTs/E_Gantry/E_GantryMachineState.TcDUT
{attribute 'strict'}
{attribute 'qualified_only'}
TYPE E_GantryMachineState :
(
	eIdle					:= 0,
	eAborting				:= 10,
	eAborted				:= 20,
	eStopping				:= 30,
	eStopped				:= 40,
	eStarting				:= 50,
	eRunning				:= 60,
	eReseting				:= 70,
	eRestarting				:= 80,
	eError					:= 1000	
);
END_TYPE

// ---- DUTs/E_LineMachineCommand.TcDUT
{attribute 'strict'}
{attribute 'qualified_only'}
TYPE E_LineMachineCommand :
(
	eAbort	  				:= 10,
	eStop	  				:= 20,
	eRun	  				:= 30,
	eReset	  				:= 40,
	eRestart 				:= 50,
	ePause					:= 60
);
END_TYPE

// ---- DUTs/E_LineMachineMode.TcDUT
{attribute 'strict'}
{attribute 'qualified_only'}
TYPE E_LineMachineMode :
(
	eUndefined				:= 0,
	eManual					:= 1,
	eMaintenance			:= 2,
	eAutomatic				:= 3,
	eSemiAutomatic			:= 4,
	eFirstFilling			:= 5,
	eEmptying				:= 6
);
END_TYPE

// ---- DUTs/E_MachineCommand.TcDUT
{attribute 'strict'}
{attribute 'qualified_only'}
TYPE E_MachineCommand :
(
	eAbort	  				:= 10,
	eStop	  				:= 20,
	eRun	  				:= 30,
	eReset	  				:= 40,
	eRestart 				:= 50
);
END_TYPE

// ---- DUTs/E_MachineMode.TcDUT
{attribute 'strict'}
{attribute 'qualified_only'}
TYPE E_MachineMode :
(
	eUndefined				:= 0,
	eManual					:= 1,
	eMaintenance			:= 2,
	eAutomatic				:= 3,
	eSemiAutomatic			:= 4,
	eFirstFilling			:= 5,
	eEmptying				:= 6
);
END_TYPE

// ---- DUTs/E_MachineState.TcDUT
{attribute 'strict'}
{attribute 'qualified_only'}
TYPE E_MachineState :
(
	eIdle					:= 0,
	eAborting				:= 10,
	eAborted				:= 20,
	eStopping				:= 30,
	eStopped				:= 40,
	eStarting				:= 50,
	eRunning				:= 60,
	eReseting				:= 70,
	eRestarting				:= 80,
	eError					:= 1000	
);
END_TYPE

// ---- DUTs/HMI/ST_MachineMode.TcDUT
TYPE ST_MachineMode :
STRUCT
	(* Operation Mode *)
	Standby			: BOOL;
	Manual			: BOOL;
	MDI				: BOOL;
	Automatic		: BOOL;
	Homing			: BOOL;

	(* Operation State *)
	Start				: BOOL;
	Stop				: BOOL;
	Reset				: BOOL;
	Error				: BOOL;

	(* Special functions *)
	DoSingleBlock	: BOOL;
	SingleBlock		: BOOL;
    FeedHold			: BOOL;
	Backward			: BOOL;
	PrgBlockIgnore	: BOOL;
	M01Stop			: BOOL;
	//BlockSearch		: ST_BlockSearch;
	//SyntaxCheck    : ST_SyntaxCheck;
	ManualMode     : ST_ManualMode;

	(* Strings *)
	ProgramName		: STRING(1024);
	MDIString		: STRING(1024);
END_STRUCT
END_TYPE

// ---- DUTs/HMI/ST_ManualMode.TcDUT
TYPE ST_ManualMode :
STRUCT
	bKeyPos : BOOL;
	bKeyNeg : BOOL;
	bKeyRapid : BOOL;
	nLogAxisNumber : UINT;
	nInc			: UINT;
	nManualTyp	: UINT;
	nSpeed : UINT;
	nHwResolution:	UDINT;    (* Handradauflösung in 0.1 um / Umdrehung *)
END_STRUCT
END_TYPE

// ---- DUTs/NCI/E_NCIOpModes.TcDUT
TYPE E_NCIOpModes :
(
	Standby := 1,
	Automatic := 2,
	MDI := 3,
	Manual :=4,
	Homing :=5
);
END_TYPE

// ---- DUTs/NCI/ST_NCIChannelState.TcDUT
TYPE ST_NCIChannelState :
STRUCT
	(* Achtung:
		=========================
		Erster Kanal ist PTP Achsen Kanal!
	*)

	(* ---------------------------------------------
	"NOT Ready"	// 0
	"Standby"	// 1 
	"Automatic"	// 2
	"MDI"			// 3
	"Manual"		// 4
	"Reference" // 5
	 ------------------------------------------------- *)
	Mode			: ARRAY[1..8] OF INT;	(* Operation Mode *)


	(* ---------------------------------------------
	"-",				// 0 "Standby"
	"Deselected",	// 1 "Standby"
	"Selected",		// 2
	"Ready",			// 3
	"Active",		// 4
	"Hold",			// 5
	"Error",			// 6
	"",				// 7
	"",				// 8
	"Preparing",	// 9
	"Clearing",		// 10
	"Starting",		// 11
	"Aborting",		// 12
	"Stopping",		// 13
	"Resuming",		// 14
	"Resetting" };	// 15
	 ------------------------------------------------- *)
	State			: ARRAY[1..8] OF INT;	(* Operation State *)
END_STRUCT
END_TYPE

// ---- DUTs/ST_AX5000Diag.TcDUT
TYPE ST_AX5000Diag :
STRUCT
(* NC-Status *)
	nNCAxisID							: UDINT;
	bOperational						: BOOL;
	bC1DError							: BOOL;
	bWcStateError						: BOOL;
	bAxisError							: BOOL;
	iAxisErrorCode						: UDINT;

(* Drive Diag *)
	strDriveType						: STRING(19);
	strMotorType						: STRING(31);
	wDriveStatus						: WORD;
	wClass1Diag							: WORD;
	stClass1Diag						: ST_AX5000_C1D;
	stDriveStatus						: ST_AX5000DriveStatus;
	stEcSlaveStateBits					: ST_EcSlaveStateBits;
	stEcSlaveState						: ST_EcSlaveState;
	bPreopToSafeOpError					: BOOL;
	bSafeOpToOpError					: BOOL;
	stCPxInvParamList					: ST_SoE_CPxInvParamList;
	iDiagNumber							: UDINT;
	stDiagNumberList					: ST_SoE_DiagNumList;
	strDiagMessage						: STRING;
END_STRUCT
END_TYPE

// ---- DUTs/ST_ChannelSignals.TcDUT
TYPE ST_ChannelSignals :
STRUCT
	DoSingleBlock: BOOL;
	SingleBlock: BOOL;
	FeedHold: BOOL;
	Backward: BOOL;
	PrgBlockIgnore: BOOL;
	M01Stop: BOOL;
END_STRUCT
END_TYPE

// ---- POUs/Programy/Hbot/AxisOnline/DUTsAxisOnline/FBsIO/ST_FBCoESetPositionOffsetIO.TcDUT
//==================================================================================================
//							Beckhoff Automation Poland
//									18.05.2018
//	Struktura zawierajaca I/O odpowiedniego bloku
//  v1.0	|| TC v 3.1.4022.16		|| - pierwsza wersja
//==================================================================================================
TYPE ST_FBCoESetPositionOffsetIO:
STRUCT
	bExecute						: BOOL;								// Rising edge executes cmd
	lrPosition						: LREAL;
	bRelative						: BOOL;
	eFeedback						: Tc2_MC2_Drive.E_PositionOffsetFeedback;
	eMemory							: Tc2_MC2_Drive.E_PositionOffsetMemory;
	bBusy							: BOOL;
	bError							: BOOL;
	udiErrorID						: UDINT;
END_STRUCT
END_TYPE

// ---- POUs/Programy/Hbot/AxisOnline/DUTsAxisOnline/FBsIO/ST_FBGetDriveRefIO.TcDUT
//==================================================================================================
//							Beckhoff Automation Poland
//									18.04.2018
//	Struktura zawierajaca I/O odpowiedniego bloku
//  v1.0	|| TC v 3.1.4022.16		|| - pierwsza wersja
//==================================================================================================
TYPE ST_FBGetDriveRefIO:
STRUCT
	bExecute						: BOOL;								// Rising edge executes cmd
	bBusy							: BOOL;								// Read/Write busy
	bError							: BOOL;								// Read/Write error
	udiErrorID						: UDINT;							// Read/Write error ID
END_STRUCT
END_TYPE

// ---- POUs/Programy/Hbot/AxisOnline/DUTsAxisOnline/FBsIO/ST_FBHoldingBrakeCtrlIO.TcDUT
//==================================================================================================
//							Beckhoff Automation Poland
//									18.05.2018
//	Struktura zawierajaca I/O odpowiedniego bloku
//  v1.0	|| TC v 3.1.4022.16		|| - pierwsza wersja
//==================================================================================================
TYPE ST_FBHoldingBrakeCtrlIO:
STRUCT
	bForceLock 						: BOOL;								// 
	bForceUnlock					: BOOL;								// 
	bBusy							: BOOL;
	bError							: BOOL; 							// General error: parameter or CoE read.
																		// If bError = TRUE and bInitialized = FALSE - error during read motor data.
																		// If bError = TRUE and bInitialized = TRUE and (iAdsErrId <> 0 or iCANopenErrId <> 0) then I2T read error
																		// If bError = TRUE and bInitialized = TRUE and iAdsErrId = 0 and iCANopenErrId = 0 then parameter error: rTorqueLimit outside permitted range rTorqueLimitLow..rTorqueLimitHigh or Empty stDriveRef
	uiAdsErrId						: UINT;								// Forwarded output FB_CoERead_ByDriveRef
	uiSecErrId						: UINT;								// Sercos Error ID for AX5000, CanOpen error ID for AX8000
END_STRUCT
END_TYPE

// ---- POUs/Programy/Hbot/AxisOnline/DUTsAxisOnline/FBsIO/ST_FBMotorMonitoringIO.TcDUT
//==================================================================================================
//							Beckhoff Automation Poland
//									21.05.2018
//	Struktura zawierajaca I/O odpowiedniego bloku
//  v1.0	|| TC v 3.1.4022.16		|| - pierwsza wersja
//==================================================================================================
TYPE ST_FBMotorMonitoringIO:
STRUCT
	bReset							: BOOL;								// Reset FB
	rTorqueLimit					: REAL		:=	500; 				// Bipolar torque limit: 0-500%, resolution 0.1%, value goes to: 16#6072 (Ch A)/ 16#6872 (Ch B)

	bError							: BOOL; 							// General error: parameter or CoE read.
																		// If bError = TRUE and bInitialized = FALSE - error during read motor data.
																		// If bError = TRUE and bInitialized = TRUE and (iAdsErrId <> 0 or iCANopenErrId <> 0) then I2T read error
																		// If bError = TRUE and bInitialized = TRUE and iAdsErrId = 0 and iCANopenErrId = 0 then parameter error: rTorqueLimit outside permitted range rTorqueLimitLow..rTorqueLimitHigh or Empty stDriveRef
	uiAdsErrId						: UINT;								// Forwarded output FB_CoERead_ByDriveRef
	uiSecErrId						: UINT;								// Sercos Error ID for AX5000, CanOpen error ID for AX8000
	bInitialized					: BOOL;								// TRUE - Motor data read without errors, so it's possible to calculate torqe and current values in metric units
	bWarning						: BOOL;								// rCurrentF > rWarningCurrent, be aware to be over permitted range
	rWarningCurrent					: REAL; 							// Continuous Stall Current - motor parameter: 16#6075 (Ch A)/ 16#6875 (Ch B); scalled: [A]
	rTorquePerc						: REAL;								// [%]
	rTorquePercMax					: REAL;								// Max [%]
	rTorque							: REAL; 							// [Nm]
	rTorqueF						: REAL;								// Filtered [Nm]
	rTorqueMax						: REAL;								// Max [Nm]
	rCurrent						: REAL; 							// [A]
	rCurrentF						: REAL;								// Filtered [A]
	rCurrentMax						: REAL;								// Max [A]
	rI2T							: REAL; 							// Thermal Motor Utilization: 16#32C1:02 (Ch A)/ 16#36C1:02 (Ch B); units: [%]
	rI2TMax							: REAL; 							// Max % Nominal
END_STRUCT
END_TYPE

// ---- POUs/Programy/Hbot/AxisOnline/DUTsAxisOnline/FBsIO/ST_FBNcSWLimitSwitchCtrlIO.TcDUT
//==================================================================================================
//							Beckhoff Automation Poland
//									18.04.2018
//	Struktura zawierajaca I/O odpowiedniego bloku
//  v1.0	|| TC v 3.1.4022.16		|| - pierwsza wersja
//==================================================================================================
TYPE ST_FBNcSWLimitSwitchCtrlIO:
STRUCT
	bRead							: BOOL;								// Read SW limit switches values and states
	bWrite							: BOOL;								// Write SW limit switches values and states
	bReset							: BOOL; 							// Not yet
// Set values
	lrSetMinPos						: LREAL;							// SW limit switch minimum
	lrSetMaxPos						: LREAL;							// SW limit switch maximum
	bSetMinMon						: BOOL;								// Enable SW limit switch minimum monitoring
	bSetMaxMon						: BOOL;								// Enable SW limit switch maximum monitoring
// Actual values	
	lrActMinPos						: LREAL;							// Actual SW limit switch minimum
	lrActMaxPos						: LREAL;							// Actual SW limit switch maximum
	bActMinMon						: BOOL;								// SW limit switch minimum monitoring state
	bActMaxMon						: BOOL;								// SW limit switch maximum monitoring stateEND_STRUCT
//	
	bBusy							: BOOL;								// Read/Write busy
	bError							: BOOL;								// Read/Write error
	udiErrorID						: UDINT;							// Read/Write error ID
END_STRUCT
END_TYPE

// ---- POUs/Programy/Hbot/AxisOnline/DUTsAxisOnline/FBsIO/ST_FBReadChannelErrorCodeIO.TcDUT
//==================================================================================================
//							Beckhoff Automation Poland
//									18.04.2018
//	Struktura zawierajaca I/O odpowiedniego bloku
//  v1.0	|| TC v 3.1.4022.16		|| - pierwsza wersja
//==================================================================================================
TYPE ST_FBReadChannelErrorCodeIO:
STRUCT
	bExecute						: BOOL;								// Rising edge executes cmd
	bBusy							: BOOL;
	bError							: BOOL; 							// General error: parameter or CoE read.
	uiAdsErrId						: UINT;								// Forwarded output FB_CoERead_ByDriveRef
	uiSecErrId						: UINT;								// Sercos Error ID for AX5000, CanOpen error ID for AX8000
	uiChannelErrorCode				: UINT;								// 603F Error code	0x603F (Ch A)/ 0x683F (Ch B) 	UINT16
	{attribute 'displaymode':='hex'}
	uiChannelErrorCodeHex			: UINT;								// 603F Error code	0x603F (Ch A)/ 0x683F (Ch B) 	UINT16
END_STRUCT
END_TYPE

// ---- POUs/Programy/Hbot/AxisOnline/DUTsAxisOnline/FBsIO/ST_FBSetPositionOffsetIO.TcDUT
//==================================================================================================
//							Beckhoff Automation Poland
//									23.05.2018
//	Struktura zawierajaca I/O odpowiedniego bloku
//  v1.1	|| TC v 3.1.4022.16		|| - zmiana nazwy struktury usuniete CoE
//  v1.0	|| TC v 3.1.4022.16		|| - pierwsza wersja
//==================================================================================================
TYPE ST_FBSetPositionOffsetIO:
STRUCT
	bExecute						: BOOL;								// Rising edge executes cmd
	lrPosition						: LREAL;
	bRelative						: BOOL;
	eFeedback						: Tc2_MC2_Drive.E_PositionOffsetFeedback;
	eMemory							: Tc2_MC2_Drive.E_PositionOffsetMemory;
	bBusy							: BOOL;
	bError							: BOOL;
	udiErrorID						: UDINT;
	uiSecErrId						: UINT;								// Sercos Error ID for AX5000, CanOpen error ID for AX8000
END_STRUCT
END_TYPE

// ---- POUs/Programy/Hbot/AxisOnline/DUTsAxisOnline/FBsIO/ST_McAxisOnlineErrorCollection.TcDUT
//==================================================================================================
//							Beckhoff Automation Poland
//									18.04.2018
//	Struktura zawierajaca wszsytkie bbledy AxisOnline
//  v1.0	|| TC v 3.1.4022.16		|| - pierwsza wersja
//==================================================================================================
TYPE ST_McAxisOnlineErrorCollection :
STRUCT
	// Error Collection
	bError							: BOOL;						// General Error flag - all error, FB, NC, drive, communication...
	bNcError						: BOOL;
	bFBError						: BOOL;						// Mc FB error
	bCommunicationError				: BOOL;						// ADS, CoE (AX8000), SoE (AX5000)...
	bDriveError						: BOOL;
	uiAdsErrorID					: UINT;						// Forwarded output FB_CoERead_ByDriveRef
	uiSecErrorID					: UINT;						// Sercos Error ID for AX5000, CanOpen error ID for AX8000
	udiErrorID						: UDINT;					// Set Position Offset FB error ID
	udiNcErrorID					: UDINT;					// Nc ErrorID
	{attribute 'displaymode':='hex'}
	udiNcErrorIDHex					: UDINT;					// Nc ErrorID
	udiFBErrorID					: UDINT;					// FB ErrorID
	{attribute 'displaymode':='hex'}
	udiFBErrorIDHex					: UDINT;					// FB ErrorID

	uiDriveErrorID					: UINT;						// 603F Error code	0x603F (Ch A)/ 0x683F (Ch B) 	UINT16
	{attribute 'displaymode':='hex'}
	uiDriveErrorIDHex				: UINT;						// 603F Error code	0x603F (Ch A)/ 0x683F (Ch B) 	UINT16
END_STRUCT
END_TYPE

// ---- POUs/Programy/Hbot/AxisOnline/DUTsAxisOnline/FBsIO/ST_McAxisStatus.TcDUT
//==================================================================================================
//							Beckhoff Automation Poland
//									24.04.2018
//	Struktura zawierajaca najwazniejsze statusy osi
//  v1.0	|| TC v 3.1.4022.16		|| - pierwsza wersja
//==================================================================================================
TYPE ST_McAxisStatus :
STRUCT
	stAxisStatus			: Tc2_MC2.ST_AxisStatus;
	sAxisName				: STRING(31);				// 
	dwAxisId				: DWORD;					// Axis ID
	bNcError				: BOOL;						// Nc Eror flag
	udiNcErrorCode			: UDINT;					// Nc axis error code
	{attribute 'displaymode':='hex'}
	udiNcErrorCodeHex		: UDINT;					// Nc axis error code - hex format
	lrActPos				: LREAL;					// Actual position (absolut value from NC)
	lrModuloActPos			: LREAL;					// Actual modulo position (absolut value from NC)
	lrActVelo				: LREAL;					// Actual velocity
	lrActAcc				: LREAL;					// Actual acceleration
	lrActTorque				: LREAL;
	lrSetPos				: LREAL;					// Set position (absolut value from NC)
	lrSetVelo				: LREAL;					// Set velocity
	lrSetAcc				: LREAL;					// Set acceleration
	lrSetTorque				: LREAL;

	lrPosDiff				: LREAL;					// Position difference (lag distance)
	bAxisReady				: BOOL;						// Axis.Status.Operational
	bHomed					: BOOL;
	bCoupled				: BOOL;
	bAcceptBlockedDrive		: BOOL;						// Force move back from limit switch
END_STRUCT
END_TYPE

// ---- POUs/Programy/Hbot/AxisOnline/DUTsAxisOnline/FBsIO/ST_MCHaltIO.TcDUT
//==================================================================================================
//							Beckhoff Automation Poland
//									18.04.2018
//	Struktura zawierajaca I/O odpowiedniego bloku
//  v1.0	|| TC v 3.1.4022.16		|| - pierwsza wersja
//==================================================================================================
TYPE ST_MCHaltIO:
STRUCT
	bExecute						: BOOL;								// Rising edge executes cmd
	lrDeceleration					: LREAL;
	lrJerk							: LREAL;
	eBufferMode						: Tc2_MC2.MC_BufferMode;
	stOptions						: Tc2_MC2.ST_MoveOptions;
	bDone							: BOOL;
	bBusy							: BOOL;
	bActive							: BOOL;
	bCommandAborted					: BOOL;
	bError							: BOOL;
	udiErrorID						: UDINT;
END_STRUCT
END_TYPE

// ---- POUs/Programy/Hbot/AxisOnline/DUTsAxisOnline/FBsIO/ST_MCHomeIO.TcDUT
//==================================================================================================
//							Beckhoff Automation Poland
//									18.04.2018
//	Struktura zawierajaca I/O odpowiedniego bloku
//  v1.0	|| TC v 3.1.4022.16		|| - pierwsza wersja
//==================================================================================================
TYPE ST_MCHomeIO:
STRUCT
	bExecute						: BOOL;								// Rising edge executes cmd
	lrPosition						: LREAL					:= DEFAULT_HOME_POSITION;
	eHomingMode						: Tc2_MC2.MC_HomingMode;
	eBufferMode						: Tc2_MC2.MC_BufferMode;
	stOptions						: Tc2_MC2.ST_HomingOptions;
	bCalibrationCam					: BOOL;
	bDone							: BOOL;
	bBusy							: BOOL;
	bActive							: BOOL;
	bCommandAborted					: BOOL;
	bError							: BOOL;
	udiErrorID						: UDINT;
END_STRUCT
END_TYPE

// ---- POUs/Programy/Hbot/AxisOnline/DUTsAxisOnline/FBsIO/ST_MCJogIO.TcDUT
//==================================================================================================
//							Beckhoff Automation Poland
//									18.04.2018
//	Struktura zawierajaca I/O odpowiedniego bloku
//  v1.0	|| TC v 3.1.4022.16		|| - pierwsza wersja
//==================================================================================================
TYPE ST_MCJogIO:
STRUCT
	bSlowForward					: BOOL;
	bSlowBackward					: BOOL;
	bFastForward					: BOOL;
	bFastBackward					: BOOL;
	bJogForward						: BOOL;
	bJogBackwards					: BOOL;
	eMode							: Tc2_MC2.E_JogMode;
	lrPosition						: LREAL;
	lrVelocity						: LREAL;
	lrAcceleration					: LREAL;
	lrDeceleration					: LREAL;
	lrJerk							: LREAL;
	bDone							: BOOL;
	bBusy							: BOOL;
	bActive							: BOOL;
	bCommandAborted					: BOOL;
	bError							: BOOL;
	udiErrorID						: UDINT;
END_STRUCT
END_TYPE

// ---- POUs/Programy/Hbot/AxisOnline/DUTsAxisOnline/FBsIO/ST_MCMoveAbsoluteIO.TcDUT
//==================================================================================================
//							Beckhoff Automation Poland
//									18.04.2018
//	Struktura zawierajaca I/O odpowiedniego bloku
//  v1.0	|| TC v 3.1.4022.16		|| - pierwsza wersja
//==================================================================================================
TYPE ST_MCMoveAbsoluteIO:
STRUCT
	bExecute						: BOOL;								// Rising edge executes cmd
	lrPosition						: LREAL;
	lrVelocity						: LREAL;
	lrAcceleration					: LREAL;
	lrDeceleration					: LREAL;
	lrJerk							: LREAL;
	eBufferMode						: Tc2_MC2.MC_BufferMode;
	stOptions						: Tc2_MC2.ST_MoveOptions;
	bDone							: BOOL;
	bBusy							: BOOL;
	bActive							: BOOL;
	bCommandAborted					: BOOL;
	bError							: BOOL;
	udiErrorID						: UDINT;
END_STRUCT
END_TYPE

// ---- POUs/Programy/Hbot/AxisOnline/DUTsAxisOnline/FBsIO/ST_MCMoveModuloIO.TcDUT
//==================================================================================================
//							Beckhoff Automation Poland
//									18.04.2018
//	Struktura zawierajaca I/O odpowiedniego bloku
//  v1.0	|| TC v 3.1.4022.16		|| - pierwsza wersja
//==================================================================================================
TYPE ST_MCMoveModuloIO:
STRUCT
	bExecute						: BOOL;								// Rising edge executes cmd
	lrPosition						: LREAL;
	lrVelocity						: LREAL;
	lrAcceleration					: LREAL;
	lrDeceleration					: LREAL;
	lrJerk							: LREAL;
	eDirection						: Tc2_MC2.MC_Direction 		:= MC_Positive_Direction; // MC_Positive_Direction := 1, MC_Shortest_Way, MC_Negative_Direction, MC_Current_Direction
	eBufferMode						: Tc2_MC2.MC_BufferMode;
	stOptions						: Tc2_MC2.ST_MoveOptions;
	bDone							: BOOL;
	bBusy							: BOOL;
	bActive							: BOOL;
	bCommandAborted					: BOOL;
	bError							: BOOL;
	udiErrorID						: UDINT;
END_STRUCT
END_TYPE

// ---- POUs/Programy/Hbot/AxisOnline/DUTsAxisOnline/FBsIO/ST_MCMoveRelativeIO.TcDUT
//==================================================================================================
//							Beckhoff Automation Poland
//									18.04.2018
//	Struktura zawierajaca I/O odpowiedniego bloku
//  v1.0	|| TC v 3.1.4022.16		|| - pierwsza wersja
//==================================================================================================
TYPE ST_MCMoveRelativeIO:
STRUCT
	bExecute						: BOOL;								// Rising edge executes cmd
	lrDistance						: LREAL;
	lrVelocity						: LREAL;
	lrAcceleration					: LREAL;
	lrDeceleration					: LREAL;
	lrJerk							: LREAL;
	eBufferMode						: Tc2_MC2.MC_BufferMode;
	stOptions						: Tc2_MC2.ST_MoveOptions;
	bDone							: BOOL;
	bBusy							: BOOL;
	bActive							: BOOL;
	bCommandAborted					: BOOL;
	bError							: BOOL;
	udiErrorID						: UDINT;
END_STRUCT
END_TYPE

// ---- POUs/Programy/Hbot/AxisOnline/DUTsAxisOnline/FBsIO/ST_MCMoveVelocityIO.TcDUT
//==================================================================================================
//							Beckhoff Automation Poland
//									18.04.2018
//	Struktura zawierajaca I/O odpowiedniego bloku
//  v1.0	|| TC v 3.1.4022.16		|| - pierwsza wersja
//==================================================================================================
TYPE ST_MCMoveVelocityIO:
STRUCT
	bExecute						: BOOL;								// Rising edge executes cmd
	lrVelocity						: LREAL;
	lrAcceleration					: LREAL;
	lrDeceleration					: LREAL;
	lrJerk							: LREAL;
	eDirection						: Tc2_MC2.MC_Direction 		:= MC_Positive_Direction; // MC_Positive_Direction := 1, MC_Shortest_Way, MC_Negative_Direction, MC_Current_Direction
	eBufferMode						: Tc2_MC2.MC_BufferMode;
	stOptions						: Tc2_MC2.ST_MoveOptions;
	bDone							: BOOL;
	bInVelocity						: BOOL;								// The same meaning as bDone
	bBusy							: BOOL;
	bActive							: BOOL;
	bCommandAborted					: BOOL;
	bError							: BOOL;
	udiErrorID						: UDINT;
END_STRUCT
END_TYPE

// ---- POUs/Programy/Hbot/AxisOnline/DUTsAxisOnline/FBsIO/ST_MCPowerIO.TcDUT
//==================================================================================================
//							Beckhoff Automation Poland
//									18.04.2018
//	Struktura zawierajaca I/O odpowiedniego bloku
//  v1.0	|| TC v 3.1.4022.16		|| - pierwsza wersja
//==================================================================================================
TYPE ST_MCPowerIO:
STRUCT
	bEnable							: BOOL;
	bEnable_Positive				: BOOL;
	bEnable_Negative				: BOOL;
	lrOverride						: LREAL := 100.0;
	eBufferMode						: Tc2_MC2.MC_BufferMode;
	stOptions						: Tc2_MC2.ST_PowerOptions;
	bStatus							: bool; // Same meaning as Done
	bBusy							: BOOL;
	bActive							: BOOL;
	bError							: BOOL;
	udiErrorID						: UDINT;
END_STRUCT
END_TYPE

// ---- POUs/Programy/Hbot/AxisOnline/DUTsAxisOnline/FBsIO/ST_MCReadDriveAddressIO.TcDUT
//==================================================================================================
//							Beckhoff Automation Poland
//									18.04.2018
//	Struktura zawierajaca I/O odpowiedniego bloku
//  v1.0	|| TC v 3.1.4022.16		|| - pierwsza wersja
//==================================================================================================
TYPE ST_MCReadDriveAddressIO:
STRUCT
	bExecute						: BOOL;								// Rising edge executes cmd
	bDone							: BOOL;
	bBusy							: BOOL;
	bError							: BOOL;
	udiErrorID						: UDINT;
END_STRUCT
END_TYPE

// ---- POUs/Programy/Hbot/AxisOnline/DUTsAxisOnline/FBsIO/ST_MCReadParameterSetIO.TcDUT
//==================================================================================================
//							Beckhoff Automation Poland
//									18.04.2018
//	Struktura zawierajaca I/O odpowiedniego bloku
//  v1.0	|| TC v 3.1.4022.16		|| - pierwsza wersja
//==================================================================================================
TYPE ST_MCReadParameterSetIO :
STRUCT
	bExecute						: BOOL;								// Rising edge executes cmd
	bDone							: BOOL;
	bBusy							: BOOL;
	bError							: BOOL;
	udiErrorID						: UDINT;
END_STRUCT
END_TYPE

// ---- POUs/Programy/Hbot/AxisOnline/DUTsAxisOnline/FBsIO/ST_MCResetIO.TcDUT
//==================================================================================================
//							Beckhoff Automation Poland
//									18.04.2018
//	Struktura zawierajaca I/O odpowiedniego bloku
//  v1.0	|| TC v 3.1.4022.16		|| - pierwsza wersja
//==================================================================================================
TYPE ST_MCResetIO:
STRUCT
	bExecute						: BOOL;								// Rising edge executes cmd
	bDone							: BOOL;
	bBusy							: BOOL;
	bError							: BOOL;
	udiErrorID						: UDINT;
END_STRUCT
END_TYPE

// ---- POUs/Programy/Hbot/AxisOnline/DUTsAxisOnline/FBsIO/ST_MCSetPositionIO.TcDUT
//==================================================================================================
//							Beckhoff Automation Poland
//									18.04.2018
//	Struktura zawierajaca I/O odpowiedniego bloku
//  v1.0	|| TC v 3.1.4022.16		|| - pierwsza wersja
//==================================================================================================
TYPE ST_MCSetPositionIO:
STRUCT
	bExecute						: BOOL;								// Rising edge executes cmd
	lrPosition						: LREAL;
	bMode							: BOOL;								// RELATIVE = True, ABSOLUTE = False (Default)
	stOptions						: Tc2_MC2.ST_SetPositionOptions;
	bDone							: BOOL;
	bBusy							: BOOL;
	bError							: BOOL;
	udiErrorID						: UDINT;
END_STRUCT
END_TYPE

// ---- POUs/Programy/Hbot/AxisOnline/DUTsAxisOnline/FBsIO/ST_MCStopIO.TcDUT
//==================================================================================================
//							Beckhoff Automation Poland
//									18.04.2018
//	Struktura zawierajaca I/O odpowiedniego bloku
//  v1.0	|| TC v 3.1.4022.16		|| - pierwsza wersja
//==================================================================================================
TYPE ST_MCStopIO:
STRUCT
	bExecute						: BOOL;								// Rising edge executes cmd
	lrDeceleration					: LREAL; 
	lrJerk							: LREAL;
	stOptions						: Tc2_MC2.ST_MoveOptions;
	bDone							: BOOL;
	bBusy							: BOOL;
	bActive							: BOOL;
	bCommandAborted					: BOOL;
	bError							: BOOL;
	udiErrorID						: UDINT;
END_STRUCT
END_TYPE

// ---- POUs/Programy/Hbot/AxisOnline/DUTsAxisOnline/ST_AX5000Diag_1.TcDUT
TYPE ST_AX5000Diag_1 :
STRUCT
(* NC-Status *)
	nNCAxisID							: UDINT;
	bOperational						: BOOL;
	bC1DError							: BOOL;
	bWcStateError						: BOOL;
	bAxisError							: BOOL;
	iAxisErrorCode						: UDINT;

(* Drive Diag *)
	strDriveType						: STRING(19);
	strMotorType						: STRING(31);
	wDriveStatus						: WORD;
	wClass1Diag							: WORD;
	stClass1Diag						: ST_AX5000_C1D;
	stDriveStatus						: ST_AX5000DriveStatus;
	stEcSlaveStateBits					: ST_EcSlaveStateBits;
	stEcSlaveState						: ST_EcSlaveState;
	bPreopToSafeOpError					: BOOL;
	bSafeOpToOpError					: BOOL;
	stCPxInvParamList					: ST_SoE_CPxInvParamList;
	iDiagNumber							: UDINT;
	stDiagNumberList					: ST_SoE_DiagNumList;
	strDiagMessage						: STRING;
END_STRUCT
END_TYPE

// ---- POUs/Programy/Hbot/AxisOnline/DUTsAxisOnline/ST_McAxisOnline.TcDUT
//==================================================================================================
//							Beckhoff Automation Poland
//									18.05.2018
//	Struktura interfejsu do obslugi Axis Online
//	v1.1	|| TC v 3.1.4022.16		|| - zmiana nazw struktur 
// 									 ST_FBCoEAX8000SetPositionOffsetIO 	--> ST_FBCoESetPositionOffsetIO
// 									 ST_FBHoldingBrakeCtrlAX8000IO 		--> ST_FBHoldingBrakeCtrlIO
// 									 ST_FBMotorMonitoringAX8000IO 		--> ST_FBMotorMonitoringIO
//  v1.0	|| TC v 3.1.4022.16		|| - pierwsza wersja
//==================================================================================================
TYPE ST_McAxisOnline :
STRUCT
	// Base administration
	mcPower							: ST_MCPowerIO;
	mcStop							: ST_MCStopIO;
	mcHalt							: ST_MCHaltIO;
	mcSS1							: ST_MCStopIO;
	mcSS2							: ST_MCStopIO;
	mcReset							: ST_MCResetIO;
	mcHome							: ST_MCHomeIO;
	mcSetPosition					: ST_MCSetPositionIO;
	stSetPositionOffset				: ST_FBSetPositionOffsetIO;
	// Base move
	mcMoveAbsolute					: ST_MCMoveAbsoluteIO;
	mcMoveRelative					: ST_MCMoveRelativeIO;
	mcMoveVelocity					: ST_MCMoveVelocityIO;
	mcMoveModulo					: ST_MCMoveModuloIO;
	mcMoveAbsolute2					: ST_MCMoveAbsoluteIO;
	mcMoveRelative2					: ST_MCMoveRelativeIO;
	mcMoveVelocity2					: ST_MCMoveVelocityIO;
	mcMoveModulo2					: ST_MCMoveModuloIO;
	mcJog							: ST_MCJogIO;
	// States, parameters, monitoring and diag
	stMotorMonitoring				: ST_FBMotorMonitoringIO;
	stHoldingBrake					: ST_FBHoldingBrakeCtrlIO;
	stNcLimitSwitch					: ST_FBNcSWLimitSwitchCtrlIO;
	stAxisParameter					: Tc2_MC2.ST_AxisParameterSet;
	stDriveRef						: Tc2_EtherCAT.ST_DriveRef;
	stDriveAddress					: Tc2_MC2.ST_DriveAddress;
	stChannelErrorCode				: ST_FBReadChannelErrorCodeIO;
	stStatus						: ST_McAxisStatus;
	// FBs
	stGetDriveRef					: ST_FBGetDriveRefIO;					// IO for FB_GetDriveRef
	mcReadDriveAddress				: ST_MCReadDriveAddressIO;				// IO for MC_ReadDriveAddress
	mcReadParameterSet				: ST_MCReadParameterSetIO;				// IO for MC_ReadParameterSet
	stError							: ST_McAxisOnlineErrorCollection;		// Error collection for all Axis Online functions
	bError							: BOOL;									// General Error flag - all error, FB, NC, drive, communication... check stError for detail
END_STRUCT
END_TYPE

// ---- GVLs/Global_HMI.TcGVL
VAR_GLOBAL
	PLCAxisEnable				: BOOL;			(* HMI -> PLC *)
	PLCMachineMode				: ARRAY[0..5] OF ST_MachineMode;
	PLCNciChannelState      	: ST_NCIChannelState;                                 (* PLC -> HMI *)
			/// HMI -> PLC 
	PLCChannelSignals			: ST_ChannelSignals;
	PLCDeleteFailure			: BOOL;			(* HMI -> PLC *)
	PLCReset					: BOOL;			(* HMI -> PLC *)
	PLCFeedOverride				: UINT := 100;			(* HMI -> PLC *)
	PLCSpindleOverride			: UINT := 100;			(* HMI -> PLC *)	
	PLCSelectedChannel			: INT:=2;				
	
	// Spindle variables
	sActiveSpindleVal			: STRING;
	sCmdSpindleVal				: STRING;
	sSpindleCurrentPos			: STRING;
	
	// Variables for the modules "InformPlc" 
	bToggle						: BOOL;
	sActualForm					: STRING[255];
	nUserLevel					: INT;
	sUserName					: STRING[255];
	bExitApp					: BOOL;
	nUserId						: UINT;
			
	
END_VAR

// ---- GVLs/GVL.TcGVL
{attribute 'qualified_only'}
VAR_GLOBAL CONSTANT
	
END_VAR
VAR_GLOBAL
	//
	bAllUnitsReady						: BOOL;					// All machine units are OK, and ready to operate
	bGeneralOK							: BOOL;					// There is no Warning, Error or Fatal Error - just when it's true - You can operate
	bGeneralWarning						: BOOL;					// Warning - just message/event - no reaction
	bGeneralError						: BOOL;					// Error - machine has to stop, start is possible from this position
	bGeneralFatalError					: BOOL;					// Fatal error causes machine stop. You have to go back for cycle begin.

	// 
	bRestartRequired					: BOOL;					// In case of fatal error, when whole process restart required
	bMuteGeneralError					: BOOL;					// Just for service/maitenance - if You are aware of consequences You can force muting mode
	bMuteGeneralFatalError				: BOOL;					// Just for service/maitenance - if You are aware of consequences You can force muting mode
END_VAR

// ---- GVLs/GVL_AXIS.TcGVL
{attribute 'qualified_only'}
VAR_GLOBAL
	//serwo kartoniarka 
		stAxis1 :AXIS_REF;
		bLogDriveDiagMsgs 	: BOOL := FALSE;
	bForceStateChgAfterDrvReset : BOOL := FALSE;
		bEnable :BOOL;
	
		//serwo kierownica 
		stAxis2 :AXIS_REF;
		//enkoder balluff 

		EC_Magazyn :AXIS_REF;	
		F_Magazyn :AXIS_REF;	
END_VAR

// ---- GVLs/GVL_EventsSimple.TcGVL
//==================================================================================================
//							Beckhoff Automation Poland
//									22.12.2016
//  v1.3	|| TC v 3.1.4020.28		|| - FIRST_MESSAGE i LAST_MESSAGE zmian typu z UDINT na DINT - znikaja ostrzezenia
//  v1.2	|| TC v 3.1.4020.28		|| - zmiana nazwy zakładki globalnych, zmiana nazwy zmiennej aAlarms na aEventsSimple
//  v1.1	|| TC v 3.1.4020.28		|| - dodanie wersjonowania: dodanie MSG_MESSAGE_List
// 	v1.0	|| TC v 3.1.4020.0		|| - pierwsza wersja
//==================================================================================================
VAR_GLOBAL CONSTANT
	FIRST_MESSAGE			: DINT := 1;
	LAST_MESSAGE			: DINT := 1200;
END_VAR
VAR_GLOBAL
	// Tablice alarmow, komunikatow i ostrzezen.
	MSG_ALARM_List			: ARRAY[FIRST_MESSAGE..LAST_MESSAGE] OF BOOL;
	MSG_WARNING_List		: ARRAY[FIRST_MESSAGE..LAST_MESSAGE] OF BOOL;
	MSG_MESSAGE_List		: ARRAY[FIRST_MESSAGE..LAST_MESSAGE] OF BOOL;
	aEventsSimple			: ARRAY[1..80] OF ST_ReadEvent;					// Tablica odczytywana przez obiekt wizualizacji Event table
END_VAR

// ---- GVLs/GVL_GLOBAL.TcGVL
{attribute 'qualified_only'}
VAR_GLOBAL
	
	bZaladowanyPrawidlo			:BOOL;//ploter zaladowal prawidlo
	bZgodaNaRuchPrawidlo        :BOOL;//zgoda na jazde plotera 
	bLadujPrawidlo				:BOOL;//zgoda na zaladowanie butelek do kartonu
	bEnableKartoniarka :BOOL;
	bEnablePloter :BOOL;
	bEnableZaklejarka :BOOL;
	bEnableKierownica :BOOL;
	Zabierz_Z_Kierownicy:BOOL;
	Ploter_pobral :BOOL;
	odloz_do_kartonu:BOOL;
	
	//kartoniarka manual
	zaw_ssawki_cewka: BOOL;
	zaw_zeby_cewka: BOOL;
	zaw_skos_cewka: BOOL;
	zaw_klap_krot_cewka: BOOL;
	zaw_klap_dlug_cewka: BOOL;
	zaw_wypychacz_cewka: BOOL;
	falownik_pasow_cewka: BOOL;
	falownik_cewka_CW_CCW: BOOL;
	
	//kartoniarka automat
	zaw_ssawki_auto: BOOL;
	S_skos: BOOL;
	S_KL_Dl: BOOL;
	S_KL1_K: BOOL;
	S_KL2_K: BOOL;
	S_Wy: BOOL;
	F1_CW: BOOL; // tutaj bylo falownik_pasow_auto
	F1_CCW: BOOL;// tego nie bylo 
	
	Error_ind_kart: BOOL;
	Error_numb_kart: INT;
	Error_reset_kart: BOOL;
	
	//ploter manual
	zaw_chwyt1_cewka: BOOL;
	zaw_chwyt2_cewka: BOOL;
	zaw_prawidlo_cewka: BOOL;
	zaw_prawidlo_dol_cewka: BOOL;
	zaw_hamulec_cewka: BOOL;
	falownik_rolek_cewka: BOOL;
	bPlotJogF :BOOL;
	bPlotJogB :BOOL;
	//ploter automat
	zaw_chwyt1_auto: BOOL;
	zaw_chwyt2_auto: BOOL;
	zaw_prawidlo_auto: BOOL;
	zaw_prawidlo_dol_auto: BOOL;
	zaw_hamulec_auto: BOOL;
	falownik_rolek_auto: BOOL;
	
	
	//kierownica manual
	zaw_ham1_kier_cewka: BOOL;
	zaw_ham2_kier_cewka: BOOL;
	serwo_kier_cewka: BOOL;
	zaw_hamulec_kier_cewka: BOOL;
	falownik_podajnik_kier_cewka: BOOL;
	
	//kierownica automat
	zaw_ham1_kier_auto: BOOL;
	zaw_ham2_kier_auto: BOOL;
	serwo_kier_auto: BOOL;
	zaw_hamulec_kier_auto: BOOL;
	falownik_podajnik_kier_auto: BOOL;
	b_FK_CW: BOOL;
	b_FK_CCW: BOOL;
	
	reset_licznik: BOOL;
	stan_licz: ARRAY[1..5] OF INT;
	Error_pakowania: BOOL;
	Error_numb_kier: INT;
	


	
	//zaklejarka manual
	sil_zamykacz_zaklejarka_cewka: BOOL;
	tasmy_zaklejarka_cewka: BOOL;
	//zaklejarka automat
	zamykacz_zaklejarka_auto: BOOL;
	bFZaklejarka_CCW: BOOL;

	
END_VAR

// ---- GVLs/GVL_HMI.TcGVL
{attribute 'qualified_only'}
VAR_GLOBAL
		bManual				:BOOL;
		bAuto				:BOOL;
		bReset				:BOOL;
		Error_ind			:BOOL;
		bAutoWybor			:BOOL;
		bEnableKartoniarka	:BOOL;
		bEnableZaklejarka	:BOOL;
		bEnablePloter		:BOOL;
		bEnableKierownica	:BOOL;
		bHmiJogF			:BOOL;
		bHmiJogB			:BOOL;
		bHmiJogKF			:BOOL;
		bHmiJogKB			:BOOL;
		bHmiJogZakCw		:BOOL;
		bHmiJogZakCCW		:BOOL;
		bHmiMagCw			:BOOL;
		bHmiMagCcw			:BOOL;
		bHmiPlotCw			:BOOL;
		bHmiPlotCCw			:BOOL;
		strona				:INT;
		strona_1			:INT;
		iFreqKartoniarkaMan :INT;
		iFreqKierownicaMan :INT;
		b_CCW_Manual_Ka_F1	 :BOOL	;// ccw manual falownik 1 
		b_CW_Manual_Ka_F1	 :BOOL	;// cw manual falownik 1 
		b_CCW_Manual_FMKart	 :BOOL	;// ccw manual falownik kartoniarka  magazyn
		b_CW_Manual_FMKart	 :BOOL	;// cw manual falownik kartoniarka  magazyn
		b_CCW_Manual_Pl_F	 :BOOL	;// ccw manual falownik ploter podajnik
		b_CW_Manual_Pl_F	 :BOOL	;// cw manual falownik ploter podajnik
		b_CCW_Manual_Kier_F	 :BOOL	;// ccw manual kierwonica podajnik
		b_CW_Manual_Kier_F	 :BOOL	;// cw manual kierwonica podajnik
		Nastepny_Karton 	 :BOOL	;// cw manual kierwonica podajnik
		A_Start				 : BOOL;
		A_Stop				 : BOOL;
		bDojkiM				 : BOOL;// dojki tryb manualny 
		iWydajnosc			:INT;//wydajnosc linii 
		INT_idError			:INT;
		J_Vel				: LREAL;
		J_VelK				: LREAL;
		zaladowalem:BOOL;
		b_Zmienna_test_in	:BOOL;
		b_zmienna_test_out :BOOL;
		//kartoniarka
		przycisk_zaw_ssawki: BOOL;
		przycisk_zaw_zeby: BOOL;
		przycisk_zaw_skos: BOOL;
		przycisk_zaw_klap_krot: BOOL;
		przycisk_zaw_klap_dlug: BOOL;
		przycisk_zaw_wypychacz: BOOL;
		przycisk_falownik_pasow: BOOL;
		przycisk_falownik_CW_CCW: BOOL;
		//ploter
		przycisk_zaw_chwyt1: BOOL;
		przycisk_zaw_chwyt2: BOOL;
		przycisk_zaw_prawidlo: BOOL;
		przycisk_zaw_prawdidlo_dol: BOOL;
		przycisk_zaw_hamulec: BOOL;
		przycisk_falownik_rolek: BOOL;
		//kierownica
		przycisk_zaw_ham1_kier: BOOL;
		przycisk_zaw_ham2_kier: BOOL;
		przycisk_serwo_kier: BOOL;
		przycisk_zaw_hamulec_kier: BOOL;
		przycisk_falownik_podajnik_kier: BOOL;
		ErrorResetKier: BOOL;
		Wymus_pobranie: BOOL;
		//zaklejarka
		przycisk_sil_zamykacz_zaklejarka: BOOL;
		przycisk_tasmy_zaklejarka: BOOL;
END_VAR
VAR_GLOBAL PERSISTENT
	Bit_Startu: BOOL := TRUE;
END_VAR
VAR_GLOBAL
		zaladuj:BOOL;
END_VAR

// ---- GVLs/GVL_IO.TcGVL
{attribute 'qualified_only'}
VAR_GLOBAL	
	
		//zmienne systemowe

		Zmienna_P_On : BOOL :=TRUE;		
		//wyjścia
		S_Zeb 		AT%Q* :BOOL	;
		S_Kl_1		AT%Q* :BOOL	;
		S_Kl_2		AT%Q* :BOOL	;
		P_Vac		AT%Q* :BOOL	;
		S_skos		AT%Q* :BOOL	;
		S_Wypych	AT%Q* :BOOL	;
		S_Fal  		AT%Q* :BOOL	;
		S_Ssawki 	AT%Q* :BOOL	;
		IOLinkCh1T	AT%Q* :BOOL	;
		IOLinkCh3T	AT%Q* :BOOL	;	
		//wejscia
		Wyp_wys	AT%I* :BOOL	;
		Wyp_cof AT%I* :BOOL	;	
		Vacuostat AT%I* :BOOL	;		// tutaj jest dodatkowo czujnik.podciś... na trojniku
		Skos_wyp AT%I*	: BOOL;
		Skos_cof AT%I* :BOOL	;
		Presostat AT%I* :BOOL	;		// tutaj dod. presostat5... czujnik cisnienia...kontrola ciśnienia
		Kl_1_wyp AT%I* :BOOL;
		Kl_1_cof AT%I* :BOOL	;
		Kl_2_wyp AT%I* :BOOL	;
		Kl_2_cof AT%I* :BOOL	;
		Zeb_Wyp AT%I* :BOOL	;
		Zeb_Cof AT%I*: BOOL;
		SI_DI AT%I* :UDINT	;
		Cz_M_D  AT%I* :BOOL	; 				//czujnik magazynu dociskowy 
		
		bRygiel  AT%I* :BOOL	; 
		bRygie2  AT%I* :BOOL	; 
		bRygie3  AT%I* :BOOL	; 
		bBezpiecznik1 AT%I* :BOOL	; 
		bBezpiecznik2 AT%I* :BOOL	; 
		bBezpiecznik3 AT%I* :BOOL	; 
		bStart AT%I* :BOOL	; 
		bStop AT%I* :BOOL	; 
		bStartGlobal AT%I* :BOOL	; 
		
		//wejscia E1008 kartoniarka 
		b1K1 AT%I* :BOOL	; //PRZYCISK start
		b1K2 AT%I* :BOOL	; 
		b1K3 AT%I* :BOOL	; //PRZYCISK stop
		b1K4 AT%I* :BOOL	; 
		b1K5 AT%I* :BOOL	; 
		b1K6 AT%I* :BOOL	;
		b1K7 AT%I* :BOOL	; 
		b1K8 AT%I* :BOOL	; //PRZYCISK reset 
		//wyjscia E2008 kartoniarka 
		
		K1K1 AT%Q* :BOOL	; 		//tylnie łapki
		K1K2 AT%Q* :BOOL	;  //lampka reset 
		K1K3 AT%Q* :BOOL	; //przednie łapki
		K1K4 AT%Q* :BOOL	; //podpych
		K1K5 AT%Q* :BOOL	; //lampka start
		K1K6 AT%Q* :BOOL	;
		K1K7 AT%Q* :BOOL	; //lampka stop
		K1K8 AT%Q* :BOOL	; 
		
		//magazyn kartońów
		
		bCzujnik_Trzymacz1 AT%I* :BOOL;
		bCzujnik_Trzymacz2 AT%I* :BOOL;
		
	
END_VAR

// ---- GVLs/GVL_IO_K.TcGVL
{attribute 'qualified_only'}
VAR_GLOBAL
	
			//wyjścia
			bK1 AT%Q* :BOOL	;	// zaw_hamulec 1
			bK2 AT%Q* :BOOL	;	// zaw_hamulec 2
			bK3 AT%Q* :BOOL	;	//  zaw hamulec
			bK4 AT%Q* :BOOL	;	//  serwo 
			bK5 AT%Q* :BOOL	;	// falownik podajnika
			bK6 AT%Q* :BOOL	;	// 
			bK7 AT%Q* :BOOL	;	// 
			bK8 AT%Q* :BOOL	;	// 
			

//wejścia
			
			b4B1 AT%I* :BOOL	; //czujnik liczenie 1
			b4B2 AT%I* :BOOL	; //czujnik liczenie 2
			b4B3 AT%I* :BOOL	; //czujnik liczenie 3
			b4B4 AT%I* :BOOL	; //czujnik liczenie 4
			b4B5 AT%I* :BOOL	; //czujnik liczenie 5
			b4B6 AT%I* :BOOL	; // kontraktron 2
			b4B7 AT%I* :BOOL	; // kontraktron 1
			b4B8 AT%I* :BOOL	; //czujnik obecności butelki
END_VAR

// ---- GVLs/GVL_IO_P.TcGVL
{attribute 'qualified_only'}
VAR_GLOBAL
	

	
			//wyjścia
			 b1K1 AT%Q* :BOOL	;	// chwytak 1 
			 b2K1 AT%Q* :BOOL	;	// chwytak 2
			 b3K1 AT%Q* :BOOL	;	// prawidlo gora
			 b4K1 AT%Q* :BOOL	;	// prawidlo dol
			 b5K1 AT%Q* :BOOL	;	// hamulec
			 b6K1 AT%Q* :BOOL	;	// falownik
			 b7K1 AT%Q* :BOOL	;	// rezerwa
			 b8K1 AT%Q* :BOOL	;	// rezerwa
			 
		

			
			//wejścia
			
			b1B1 AT%I* :BOOL	; //kontraktron hamulec 1
			b2B1 AT%I* :BOOL	; //kontraktron podajnik 2
			b3B1 AT%I* :BOOL	; //czujnik hamulec  ?????? sprawdzić co to jest
			b4B1 AT%I* :BOOL	; //rezerwa
			b5B1 AT%I* :BOOL	; //kontraktron hamulec 2 
			b6B1 AT%I* :BOOL	; //kontraktron podajnik 1 
			b7B1 AT%I* :BOOL	; //rezerwa 
			b8B1 AT%I* :BOOL	; //rezerwa 
END_VAR

// ---- GVLs/GVL_Kolumna.TcGVL
{attribute 'qualified_only'}
VAR_GLOBAL
	Segment_1 AT %Q* :BYTE;
	Segment_2 AT %Q* :BYTE;
END_VAR

// ---- GVLs/GVL_Machine.TcGVL
{attribute 'qualified_only'}
VAR_GLOBAL
	eMode									: E_MachineMode := E_MachineMode.eAutomatic;	// Global machine mode
																						(*	eUndefined				:= 0,
																							eManual					:= 1,
																							eMaintenance			:= 2,
																							eAutomatic				:= 3,
																							eSemiAutomatic			:= 4,
																							eFirstFilling			:= 5,
																							eEmptying				:= 6	*)
																							
	eCommand								: E_MachineCommand; 							// Global machine command
																						(*	eAbort	  				:= 10,
																							eStop	  				:= 20,
																							eRun 	  				:= 30,
																							eReset	  				:= 40	*)
																							
	eState									: E_MachineState; 								// Global machine state
																						(*	eIdle					:= 0,
																							eAborting				:= 10,
																							eAborted				:= 20,
																							eStopping				:= 30,
																							eStopped				:= 40,
																							eStarting				:= 50,
																							eRunning				:= 60,
																							eReseting				:= 70,
																							eError					:= 1000	*)
	bNciFeedHold				: BOOL;
	bNciStart					: BOOL;
	bNCiStop					: BOOL;
																							
END_VAR

// ---- GVLs/GVL_MachineMaintenance.TcGVL
{attribute 'qualified_only'}
VAR_GLOBAL
	eMode									: E_LineMachineMode;	// Global machine mode
																						(*	eUndefined				:= 0,
																							eManual					:= 1,
																							eMaintenance			:= 2,
																							eAutomatic				:= 3,
																							eSemiAutomatic			:= 4,
																							eFirstFilling			:= 5,
																							eEmptying				:= 6	*)
																							
	eCommand								: E_LineMachineCommand; 							// Global machine command
																						(*	eAbort	  				:= 10,
																							eStop	  				:= 20,
																							eRun 	  				:= 30,
																							eReset	  				:= 40	*)
																							
	eState									: E_CaseCloserMachineState; 								// Global machine state
																						(*	eIdle					:= 0,
																							eAborting				:= 10,
																							eAborted				:= 20,
																							eStopping				:= 30,
																							eStopped				:= 40,
																							eStarting				:= 50,
																							eRunning				:= 60,
																							eReseting				:= 70,
																							eError					:= 1000	*)
																							
																							
END_VAR

// ---- GVLs/GVL_NCI.TcGVL
VAR_GLOBAL
	arrNCToPLC_NCIChannel_REF		AT %I*: ARRAY [1..nMaxNumberOfNciChannels] OF NCTOPLC_NCICHANNEL_REF;
	arrPLCToNC_NCIChannel_REF		AT %Q*: ARRAY [1..nMaxNumberOfNciChannels] OF PLCTONC_NCICHANNEL_REF;
	
	arrAxisCalibrationCam :			ARRAY [1..nMaxNumberOfAxis] OF BOOL;
	bMFunc:	 						ARRAY [1..nMaxNumberOfNciChannels,0..159] OF BOOL; (* M-Functions to acknowledge for every channel *)
	bQuitMFunc:						ARRAY [1..nMaxNumberOfNciChannels,0..159] OF BOOL; (* Array to acknolewdge M-Funktion *)
	bFastMFunc: 					ARRAY [1..nMaxNumberOfNciChannels,0..159] OF BOOL; (* fast M-Functions for every channel *)
	nGroup: 						ARRAY [1..nMaxNumberOfNciChannels] OF UDINT;  (* which logical GroupId belongs to the channel *)
	bGroup1: 						BOOL:=FALSE;
	nRParamRead:					ARRAY [1..nMaxNumberOfNciChannels, nStartIndexReadRParam..nEndIndexReadRParam] OF LREAL;	(* elements of RParam are read every second *)
	nRParamWrite:					ARRAY [1..nMaxNumberOfNciChannels, nStartIndexWriteRParam..nEndIndexWriteRParm] OF LREAL;	(* elements of RParam are write every second *)
END_VAR

(* after changing this, it is neccessary to create new links to axis and channel variables in TwinCAT SystemManager *)
VAR_GLOBAL CONSTANT
	nChan					:	UINT :=2;
	nMaxNumberOfAxis: 				UINT := 2;
	nMaxNumberOfNciChannels:		UINT := 1;  	(* channel 1 always is PTP channel, here are the maximum numbers of NCI channels is configured *)
	
	nStartIndexReadRParam:			UINT := 0;		(* Index for nRParamRead *)
	nEndIndexReadRParam:			UINT := 9;
	nStartIndexWriteRParam:			UINT := 10;		(* Index for nRParamWrite *)
	nEndIndexWriteRParm:			UINT := 29;

   	MaxNciTool:						INT := 5;(* Max.Anzahl Werkzeuge in der NCI-Verwaltung *)
END_VAR

// ---- GVLs/GVL_Omron.TcGVL
{attribute 'qualified_only'}
VAR_GLOBAL
	//Kartoniarka 
	wOmron_1_Status 	AT%I* 	:WORD;
	iOmronErectorAcc    AT%I*	:UDINT;
	iOmronErectorDcc    AT%I*	:UDINT;
	iOmron_1_ActVelo	AT%I*	:INT;
 	wOmron_1_Control	AT%Q*	:WORD;
	iOmron_1_SeVelo		AT%Q*	:INT;

	

	//Zaklejarka
	wOmron_Za_Status 	AT%I* 	:WORD; 
	iOmron_Za_ActVelo	AT%I*	:INT;	
 	wOmron_Za_Control	AT%Q*	:WORD;
	iOmron_Za_SeVelo	AT%Q*	:INT;
	
	//Ploter
	wOmron_Pl_Status 	AT%I* 	:WORD; 
	iOmron_Pl_ActVelo	AT%I*	:INT;	
 	wOmron_Pl_Control	AT%Q*	:WORD;
	iOmron_Pl_SeVelo	AT%Q*	:INT;
	
	//Kierownica
	wOmron_Kier_Status 	AT%I* 	:WORD; 
	iOmron_Kier_ActVelo	AT%I*	:INT;	
 	wOmron_Kier_Control	AT%Q*	:WORD;
	iOmron_Kier_SeVelo	AT%Q*	:INT;
END_VAR

// ---- GVLs/GVL_Recipe.TcGVL
{attribute 'qualified_only'}
VAR_GLOBAL
	

			sName : STRING;
			szer_kartonu :LREAL;
			dl_kartonu :LREAL;
			wys_kartonu :LREAL;
			
			Poz_Z_Pobranie :LREAL;
			Poz_Z_Odlozenie :LREAL;
			Poz_X_Pobranie :LREAL;
			Poz_X_Odlozenie :LREAL;
			
			Predk_plot_pobranie :LREAL;
			Predk_plot_odlozenie :LREAL;
			Predk_plot_ruch: LREAL;
			Predk_mag_pobranie :LREAL;
			Predk_mag_odlozenie :LREAL;
			
			Il_rzedow: INT;
			Il_kolumn: INT;
			
END_VAR

// ---- GVLs/GVL_RecipeTable.TcGVL
VAR_GLOBAL
	aRecipeNames 			: ARRAY[0..cMaxTableRows] OF STRING;
	aVariableNames 			: ARRAY[0..cMaxTableRows] OF STRING;
	aCurrentVariableNames 	: ARRAY[0..cMaxTableRows] OF STRING;
	aVariableValues 		: ARRAY[0..cMaxTableRows] OF STRING;
	aCurrentValues			: ARRAY[0..cMaxTableRows] OF LREAL;
	nVariableIndex			: INT;
	nVariableIndex1			: INT;
	nVariableCount 			: INT;
	nRecipeIndex 			: INT;
	nRecipeSelectionIndex 	: INT := -1;
	nRecipeCount 			: INT;
END_VAR
VAR_GLOBAL CONSTANT
	cMaxTableRows 			: INT := 14;
END_VAR

// ---- GVLs/GVL_SafetyFrom_RT2.TcGVL
{attribute 'qualified_only'}
VAR_GLOBAL
	// =================== SAFETY ===================
	bSAFETY_Error				AT %I*	: BOOL;
	bSAFETY_ResetCMD 			AT %Q*	: BOOL;
	bSAFETY_ResetBusy			AT %I*	: BOOL;
	bSAFETY_PermissionSS1		AT %I*	: BOOL; 				// Sygnal NC - TRUE - pozwolenie na prace
	bSAFETY_PermissionSS2		AT %I*	: BOOL; 				// Sygnal NC - TRUE - pozwolenie na prace
	bSAFETY_ServoKierPermitionOutSS1		AT%I* 	: BOOL;
	bSAFETY_FalownikKierPermitionOutSS1		AT%I* 	: BOOL;
	bSAFETY_ZaklejarkaKierPermitionOutSS1	AT%I* 	: BOOL;
// ======== Error and states collection =========
	dwGroupErrors				AT %I*	: DWORD;				// Group Error collection - Communication, FB, Other...
END_VAR

// ---- GVLs/GVL_Zak_IO.TcGVL
{attribute 'qualified_only'}
VAR_GLOBAL
		//wyjscia
		b_Sil_Zamkniecie AT%Q* :BOOL	;//silnik zamykakacza klapy górnej
		b_tasma AT%Q* :BOOL	;			//taśma
		bK3 AT%Q* :BOOL	;//rezerwa
		bK4 AT%Q* :BOOL	;//rezerwa
		bK5 AT%Q* :BOOL	;//rezerwa
		bK6 AT%Q* :BOOL	;//rezerwa
		bK7 AT%Q* :BOOL	;//rezerwa
		bK8 AT%Q* :BOOL	;//rezerwa
		
		
		//wejscia
		b_Czujnik_Karton	AT%I* :BOOL	;//czujnik kartonu 
		b_czujnik_OT		AT%I* :BOOL	;//czujnik obecności taśmy 
		b_kZamykacz1		AT%I* :BOOL	;//kontraktron zamykacz 1 
		b_kZamykacz2		AT%I* :BOOL	;//kontraktron zamykacz 2  
		b5B1 AT%I* :BOOL	; //rezerwa 
		b6B1 AT%I* :BOOL	; //rezerwa 
		b7B1 AT%I* :BOOL	; //rezerwa 
		b8B1 AT%I* :BOOL	; //rezerwa 
END_VAR

// ---- POUs/Programy/MAIN.TcPOU
PROGRAM MAIN
VAR
	przycisk_1 :FB_Button;
	bWritePersistent: BOOL;
	fbWritePersistentData: FB_WritePersistentData;
	nValueInt 	: INT;
	op :ARRAY[0..10] OF TOF;
	byByte_0 AT%I* :BYTE;
	byByte_1 AT%I* :BYTE;
	byByte_2 AT%I* :BYTE;
	byByte_3 AT%I* :BYTE;
	dwCounterValue AT%Q* :DWORD;
//recepty 
	nValueDword : DWORD;
	fValueReal 	: REAL;
	
	sRecipe 	: STRING;
	manual: INT;
	bManual: BOOL;

	fbBUTTONZPodajnik: FB_Button;
	dupa: BOOL;
	dupa1: BOOL;
		//kartoniarka
		zaw_ssawki: FB_BUTTON;
		zaw_skos: FB_BUTTON;
		zaw_zeby: FB_BUTTON;
		zaw_klap_krot: FB_BUTTON;
		zaw_klap_dlug: FB_BUTTON;
		zaw_wypychacz: FB_BUTTON;
		falownik_pasow: FB_BUTTON;
		falownik_CW_CCW: FB_BUTTON;
		//ploter
		zaw_chwyt1: FB_BUTTON;
		zaw_chwyt2: FB_BUTTON;
		zaw_prawidlo: FB_BUTTON;
		zaw_prawidlo_dol: FB_BUTTON;
		zaw_hamulec: FB_BUTTON;
		falownik_rolek: FB_BUTTON;
		
		//kierownica
		zaw_ham1_kier: FB_BUTTON;
		zaw_ham2_kier: FB_BUTTON;
		serwo_kier: FB_BUTTON;
		zaw_hamulec_kier: FB_BUTTON;
		falownik_podajnik_kier: FB_BUTTON;
		
		//zaklejarka
		sil_zamykacz_zaklejarka: FB_BUTTON;
		tasmy_zaklejarka: FB_BUTTON;
		//kolumna
		eColumnState 		:E_ColumState;
		
	xStartMode: BOOL;
	xGenError: BOOL;
END_VAR

VAR PERSISTENT
	bTest: BOOL;
END_VAR

// kinematyka

dwCounterValue := F_4BYTES_TO_DWORD(BByte0:=byByte_2 , BByte1:=byByte_3 , BByte2:=byByte_0 , BByte3:= byByte_1);


P_ModeStateManager();
P_Hbot_V3(eMachineMode:=GVL_Machine.eMode , eMachineCommand:=GVL_Machine.eCommand , eMachineState=>GVL_Machine.eState , bError=> );
IF  GVL_Machine.eState = E_MachineState.eRunning THEN
	bTest := TRUE;
ELSE;
	bTest:= FALSE;
END_IF
(*
PRG_HBotv2(
	bBuildHBot:= , 
	bCleanHBot:= , 
	bStopHBot:= , 
	bManualEnableHBot:= , 
	bManualDisableHbot:= , 
	bSafetyPermission:=	GVL_SafetyFrom_RT2.bSAFETY_PermissionSS1 , 
	bHbotReady=> , 
	bHbotStoper=> );
	*)
fbWritePersistentData(
	NETID:= , 
	PORT:= , 
	START:=bWritePersistent , 
	TMOUT:= , 
	MODE:= , 
	BUSY=> , 
	ERR=> , 
	ERRID=> );

	
	
//Zaklejarka
PRG_Zaklejarka();
//program kartoniarka 
PRG_Kartoniarka();
//program kierwonica
PRG_Kierownica();

//recepty 
RecipeManagement();
A_Obsluga();
//eventy
P_EventsSimple();
//przyciski
A_Przyciski();

ACTION A_Kolumna:

	(*------------------bezpieczeństwo skasowane/manual mode------------------*)
		IF GVL_SafetyFrom_RT2.bSAFETY_PermissionSS1 AND GVL_SafetyFrom_RT2.bSAFETY_PermissionSS2 AND NOT GVL_HMI.bAutoWybor AND NOT xGenError THEN
		GVL_Kolumna.Segment_1:=51;
		GVL_Kolumna.Segment_2:=3;
		eColumnState:=E_ColumState.eManualMode;
		ELSE
		eColumnState:=E_ColumState.eSafety_Ready;
		GVL_Kolumna.Segment_1:=68;
		GVL_Kolumna.Segment_2:=4;
		END_IF
	(*--------------------------Gotowy do startu/pauza----------------------*)

		IF GVL_SafetyFrom_RT2.bSAFETY_PermissionSS1 AND GVL_SafetyFrom_RT2.bSAFETY_PermissionSS2 AND GVL_HMI.bAutoWybor AND NOT xStartMode AND NOT xGenError  THEN
		GVL_Kolumna.Segment_1:=153;
		GVL_Kolumna.Segment_2:=9;
		eColumnState:=E_ColumState.eReadyToWork;
		END_IF
	(*------------------------------Pracuje----------------------*)
	
		IF GVL_SafetyFrom_RT2.bSAFETY_PermissionSS1 AND GVL_SafetyFrom_RT2.bSAFETY_PermissionSS2 AND GVL_HMI.bAutoWybor AND xStartMode AND NOT xGenError  THEN
		GVL_Kolumna.Segment_1:=17;
		GVL_Kolumna.Segment_2:=1;
		eColumnState:=E_ColumState.eWork;
		END_IF
		
	(*------------------------------obsługa przycisków start stop----------------------*)
		IF GVL_IO.B1K1 THEN
		xStartMode:=TRUE;
		ELSIF GVL_IO.B1K3 THEN
		xStartMode:=FALSE;
		END_IF
END_ACTION

ACTION A_Obsluga:
//PLOTER MANUAL 

IF GVL_HMI.bManual=TRUE AND GVL_HMI.bAuto=FALSE THEN
	

GVL_IO_P.b1K1:=gvl_hmi.bDojkiM;
//PRG_HBotv2.bManualEnableHBot:=TRUE;


ELSE
	
//PRG_HBotv2.bManualEnableHBot:=FALSE;

END_IF
//PLOTER AUTOMAT MANUAL 
IF GVL_HMI.bManual=FALSE AND GVL_HMI.bAuto=TRUE AND GVL_HMI.bEnablePloter=TRUE THEN

	
//PRG_HBotv2.bBuildHBot:=TRUE;

ELSE
	
//PRG_HBotv2.bBuildHBot:=FALSE;

END_IF
//KARTONIARKA AUTOMAT MANUAL 
IF GVL_HMI.bManual=FALSE AND GVL_HMI.bAuto=TRUE AND GVL_HMI.bEnableKartoniarka=TRUE THEN
	
GVL_GLOBAL.bEnableKartoniarka:=TRUE;

ELSE
	
GVL_GLOBAL.bEnableKartoniarka:=FALSE;

END_IF
//ZAKLEJARKA AUTOMAT MANUAL 
IF GVL_HMI.bManual=FALSE AND GVL_HMI.bAuto=TRUE AND GVL_HMI.bEnableZaklejarka=TRUE THEN
	
GVL_GLOBAL.bEnableZaklejarka:=TRUE;

ELSE
	
GVL_GLOBAL.bEnableZaklejarka:=FALSE;

END_IF
//KIEROWNCICA AUTOMAT MANUAL 
IF GVL_HMI.bManual=FALSE AND GVL_HMI.bAuto=TRUE AND GVL_HMI.bEnableKierownica=TRUE THEN
	
GVL_GLOBAL.bEnableKierownica:=TRUE;

ELSE
	
GVL_GLOBAL.bEnableKierownica:=FALSE;

END_IF


//WYBÓR AUTO MANUAL

IF gvl_hmi.bAutoWybor=TRUE THEN
	
GVL_HMI.bManual:=FALSE;
GVL_HMI.bAuto:=TRUE;
ELSE 
	
GVL_HMI.bManual:=TRUE;
GVL_HMI.bAuto:=FALSE;
END_IF
END_ACTION

ACTION A_Przyciski:
 GVL_SafetyFrom_RT2.bSAFETY_ResetCMD :=gvl_io.b1K8;//reset bezpieczenstwa
 
 IF GVL_SafetyFrom_RT2.bSAFETY_PermissionSS1=TRUE AND GVL_SafetyFrom_RT2.bSAFETY_PermissionSS2=TRUE THEN
	 
  gvl_io.K1K2:=0;
 ELSE
	 
 gvl_io.K1K2:=1;
 
 
 END_IF
 
//IF GVL_HMI.bAutoWybor=FALSE THEN 
	
//kartoniarka
zaw_ssawki(bprzyciskIn:= GVL_HMI.przycisk_zaw_ssawki,bAuto:=GVL_HMI.bAutoWybor, bprzyciskOut=>GVL_GLOBAL.zaw_ssawki_cewka);
zaw_skos(bprzyciskIn:= GVL_HMI.przycisk_zaw_skos,bAuto:=GVL_HMI.bAutoWybor, bprzyciskOut=>GVL_GLOBAL.zaw_skos_cewka);
zaw_zeby(bprzyciskIn:= GVL_HMI.przycisk_zaw_zeby,bAuto:=GVL_HMI.bAutoWybor, bprzyciskOut=>GVL_GLOBAL.zaw_zeby_cewka);
zaw_klap_krot(bprzyciskIn:= GVL_HMI.przycisk_zaw_klap_krot,bAuto:=GVL_HMI.bAutoWybor, bprzyciskOut=> GVL_GLOBAL.zaw_klap_krot_cewka);
zaw_klap_dlug(bprzyciskIn:= GVL_HMI.przycisk_zaw_klap_dlug,bAuto:=GVL_HMI.bAutoWybor, bprzyciskOut=> GVL_GLOBAL.zaw_klap_dlug_cewka);
zaw_wypychacz(bprzyciskIn:=GVL_HMI.przycisk_zaw_wypychacz,bAuto:=GVL_HMI.bAutoWybor, bprzyciskOut=>GVL_GLOBAL.zaw_wypychacz_cewka);
falownik_pasow(bprzyciskIn:= GVL_HMI.przycisk_falownik_pasow,bAuto:=GVL_HMI.bAutoWybor, bprzyciskOut=> GVL_GLOBAL.falownik_pasow_cewka);
//END_IF

IF GVL_HMI.bAuto=FALSE  AND gvl_hmi.bEnableKartoniarka=TRUE THEN 
GVL_IO.P_Vac:=GVL_GLOBAL.zaw_ssawki_cewka;
GVL_IO.S_skos:=GVL_GLOBAL.zaw_skos_cewka;
GVL_IO.S_Zeb:=GVL_GLOBAL.zaw_zeby_cewka;
GVL_IO.S_Kl_1:=GVL_GLOBAL.zaw_klap_krot_cewka;
GVL_IO.S_Kl_2:=GVL_GLOBAL.zaw_klap_dlug_cewka;
GVL_IO.S_Wypych:=GVL_GLOBAL.zaw_wypychacz_cewka;
GVL_IO.S_Fal:=GVL_GLOBAL.falownik_pasow_cewka;

END_IF

IF GVL_HMI.bAuto=TRUE THEN
GVL_IO.P_Vac :=GVL_global.zaw_ssawki_auto;
GVL_IO.S_skos:=GVL_GLOBAL.S_skos;
GVL_IO.S_Zeb:=GVL_GLOBAL.S_KL_Dl;
GVL_IO.S_Kl_1:=	GVL_global.S_KL1_K;
GVL_IO.S_Kl_2:= GVL_global.S_KL2_K;
GVL_IO.S_Wypych:= GVL_global.S_Wy;
GVL_IO.S_Fal:=GVL_GLOBAL.F1_CW; //GVL_GLOBAL.falownik_pasow_auto
END_IF

//ploter
zaw_chwyt1(bprzyciskIn:= GVL_HMI.przycisk_zaw_chwyt1,bAuto:=GVL_HMI.bAutoWybor, bprzyciskOut=>GVL_GLOBAL.zaw_chwyt1_cewka);
zaw_chwyt2(bprzyciskIn:= GVL_HMI.przycisk_zaw_chwyt2,bAuto:=GVL_HMI.bAutoWybor, bprzyciskOut=> GVL_GLOBAL.zaw_chwyt2_cewka);
zaw_prawidlo(bprzyciskIn:= GVL_HMI.przycisk_zaw_prawidlo,bAuto:=GVL_HMI.bAutoWybor, bprzyciskOut=> GVL_GLOBAL.zaw_prawidlo_cewka);
zaw_prawidlo_dol(bprzyciskIn:= GVL_HMI.przycisk_zaw_prawdidlo_dol,bAuto:=GVL_HMI.bAutoWybor, bprzyciskOut=> GVL_GLOBAL.zaw_prawidlo_dol_cewka);
zaw_hamulec(bprzyciskIn:=GVL_HMI.przycisk_zaw_hamulec,bAuto:=GVL_HMI.bAutoWybor, bprzyciskOut=>GVL_GLOBAL.zaw_hamulec_cewka);
falownik_rolek(bprzyciskIn:= GVL_HMI.przycisk_falownik_rolek,bAuto:=GVL_HMI.bAutoWybor, bprzyciskOut=> GVL_GLOBAL.falownik_rolek_cewka);

IF GVL_HMI.bAuto=FALSE AND gvl_hmi.bEnablePloter=TRUE THEN  
GVL_IO_P.b1K1:=GVL_GLOBAL.zaw_chwyt1_cewka;
GVL_IO_P.b2K1:=GVL_GLOBAL.zaw_chwyt2_cewka;
GVL_IO_P.b3K1:=GVL_GLOBAL.zaw_prawidlo_cewka;
GVL_IO_P.b4K1:=GVL_GLOBAL.zaw_prawidlo_dol_cewka;
GVL_IO_P.b5K1:=GVL_GLOBAL.zaw_hamulec_cewka;
GVL_IO_P.b6K1:=GVL_GLOBAL.falownik_rolek_cewka;
END_IF

IF GVL_HMI.bAuto=TRUE THEN
GVL_IO_P.b1K1:=GVL_GLOBAL.zaw_chwyt1_auto;
GVL_IO_P.b2K1:=GVL_GLOBAL.zaw_chwyt2_auto;
GVL_IO_P.b3K1:=GVL_GLOBAL.zaw_prawidlo_auto;
GVL_IO_P.b4K1:=GVL_GLOBAL.zaw_prawidlo_dol_auto;
GVL_IO_P.b5K1:=GVL_GLOBAL.zaw_hamulec_auto;
GVL_IO_P.b6K1:=GVL_GLOBAL.falownik_rolek_auto; 
END_IF

//kierownica
zaw_ham1_kier(bprzyciskIn:= GVL_HMI.przycisk_zaw_ham1_kier,bAuto:=GVL_HMI.bAutoWybor, bprzyciskOut=>GVL_GLOBAL.zaw_ham1_kier_cewka);
zaw_ham2_kier(bprzyciskIn:= GVL_HMI.przycisk_zaw_ham2_kier,bAuto:=GVL_HMI.bAutoWybor, bprzyciskOut=> GVL_GLOBAL.zaw_ham2_kier_cewka);
serwo_kier(bprzyciskIn:= GVL_HMI.przycisk_serwo_kier,bAuto:=GVL_HMI.bAutoWybor, bprzyciskOut=> GVL_GLOBAL.serwo_kier_cewka);
zaw_hamulec_kier(bprzyciskIn:=GVL_HMI.przycisk_zaw_hamulec_kier,bAuto:=GVL_HMI.bAutoWybor, bprzyciskOut=>GVL_GLOBAL.zaw_hamulec_kier_cewka);
falownik_podajnik_kier(bprzyciskIn:= GVL_HMI.przycisk_falownik_podajnik_kier,bAuto:=GVL_HMI.bAutoWybor, bprzyciskOut=> GVL_GLOBAL.falownik_podajnik_kier_cewka);


IF GVL_HMI.bAuto=FALSE AND gvl_hmi.bEnableKierownica=TRUE THEN 
GVL_IO_K.bK1:=GVL_GLOBAL.zaw_ham1_kier_cewka;
GVL_IO_K.bK2:=GVL_GLOBAL.zaw_ham2_kier_cewka;
GVL_IO_K.bK3:=GVL_GLOBAL.serwo_kier_cewka;
GVL_IO_K.bK4:=GVL_GLOBAL.zaw_hamulec_kier_cewka;
GVL_IO_K.bK5:=GVL_GLOBAL.falownik_podajnik_kier_cewka;
END_IF

IF GVL_HMI.bAuto=TRUE THEN
GVL_IO_K.bK1:=GVL_IO_K.bK1;
GVL_IO_K.bK2:=GVL_IO_K.bK2;
GVL_IO_K.bK4:=GVL_GLOBAL.zaw_hamulec_kier_auto;
GVL_IO_K.bK5:=GVL_GLOBAL.b_FK_CCW;
END_IF
	


//zaklejarka
sil_zamykacz_zaklejarka(bprzyciskIn:= GVL_HMI.przycisk_sil_zamykacz_zaklejarka, bAuto:=GVL_HMI.bAutoWybor,bprzyciskOUT=>GVL_GLOBAL.sil_zamykacz_zaklejarka_cewka);
tasmy_zaklejarka(bprzyciskIn:= GVL_HMI.przycisk_tasmy_zaklejarka,bAuto:=GVL_HMI.bAutoWybor, bprzyciskOUT=>GVL_GLOBAL.tasmy_zaklejarka_cewka);

IF GVL_HMI.bAuto=FALSE AND gvl_hmi.bEnableZaklejarka=TRUE THEN 
	
GVL_ZAK_IO.b_Sil_Zamkniecie:= GVL_GLOBAL.sil_zamykacz_zaklejarka_cewka;
GVL_ZAK_IO.b_tasma:= GVL_GLOBAL.tasmy_zaklejarka_cewka ;

END_IF

IF GVL_HMI.bAuto=TRUE THEN 
	
GVL_ZAK_IO.b_Sil_Zamkniecie:=GVL_GLOBAL.zamykacz_zaklejarka_auto;
GVL_ZAK_IO.b_tasma:=GVL_GLOBAL.bFZaklejarka_CCW;


ELSE
//kartoniarka
GVL_HMI.przycisk_zaw_ssawki							:=0;
GVL_HMI.przycisk_zaw_klap_krot						:=0;
GVL_HMI.przycisk_zaw_skos							:=0;
GVL_HMI.przycisk_zaw_zeby							:=0;
GVL_HMI.przycisk_zaw_klap_dlug						:=0;
GVL_HMI.przycisk_zaw_wypychacz						:=0;
GVL_HMI.przycisk_falownik_pasow						:=0;
//ploter
GVL_HMI.przycisk_zaw_chwyt1							:=0;
GVL_HMI.przycisk_zaw_chwyt2							:=0;
GVL_HMI.przycisk_zaw_prawidlo						:=0;
GVL_HMI.przycisk_zaw_prawdidlo_dol					:=0;
GVL_HMI.przycisk_zaw_hamulec						:=0;
GVL_HMI.przycisk_falownik_rolek						:=0;
//kierownica
GVL_HMI.przycisk_zaw_ham1_kier						:=0;
GVL_HMI.przycisk_zaw_ham2_kier						:=0;
GVL_HMI.przycisk_serwo_kier							:=0;
GVL_HMI.przycisk_zaw_hamulec_kier					:=0;
GVL_HMI.przycisk_falownik_podajnik_kier				:=0;
//zaklejarka
GVL_HMI.przycisk_sil_zamykacz_zaklejarka			:=0;
GVL_HMI.przycisk_tasmy_zaklejarka					:=0;
END_IF

(*Tymczasowe obsługa serwa w manualu
IF GVL_HMI.bAuto=FALSE THEN			
	J_Vel:=100;
	bJog_F:=GVL_HMI.bHmiJogKF;
	bJog_B:=GVL_HMI.bHmiJogKB;	

END_IF
*)
END_ACTION

END_PROGRAM

// ---- POUs/FB/FB_Button.TcPOU
FUNCTION_BLOCK FB_Button
VAR_INPUT
	bprzyciskIn :BOOL;
	bAuto		:BOOL;
	
END_VAR
VAR_OUTPUT
	bprzyciskOut :BOOL;
END_VAR
VAR
	zbocze	:R_TRIG;
	thne: INT;
END_VAR


zbocze(CLK:=bprzyciskIn);
IF bAuto = TRUE THEN
	
bprzyciskOut:=FALSE;
	
END_IF

IF zbocze.Q=TRUE AND bprzyciskOut=TRUE  THEN 
	
bprzyciskOut:=FALSE;

ELSIF zbocze.Q=TRUE AND bprzyciskOut=FALSE  THEN


bprzyciskOut:=TRUE;

END_IF

END_FUNCTION_BLOCK

// ---- POUs/FB/F_4BYTES_TO_DWORD.TcPOU
FUNCTION F_4BYTES_TO_DWORD : DWORD
VAR_INPUT
	BByte0		: BYTE;
	BByte1		: BYTE;
	BByte2		: BYTE;
	BByte3		: BYTE;
END_VAR
VAR
END_VAR

F_4BYTES_TO_DWORD := BByte3 *16#1000000 + BByte2 *16#10000 + BByte1 *16#100 + BByte0;

END_FUNCTION

// ---- POUs/Programy/Hbot/P_ModeStateManager.TcPOU
//==================================================================================================
//							Beckhoff Automation Poland
//									03.01.2018
//	Zarzadzeni trybami pracy i komendami - Satate Machine
// 	v1.1	|| TC v 3.1.4022.4		|| - Aktualizacja - dodano test Abort z HMI 
// 	v1.0	|| TC v 3.1.4022.4		|| - Pierwsza wersja
//==================================================================================================
PROGRAM P_ModeStateManager
VAR
	//	GVL_Machine - HMI handling
	bHMIModeRequest_Automatic			: BOOL;
	bHMIModeRequest_Manual				: BOOL;
	bHMIModeRequest_Maintenance			: BOOL;
	
	bHMICommandRequest_Run				: BOOL;
	bHMICommandRequest_Stop				: BOOL;
	bHMICommandRequest_Reset			: BOOL;
	bHMICommandRequest_Restart			: BOOL;
	bHMICommandRequest_Abort			: BOOL;
	// Rising edge detection
	rtButtonAutomatic					: R_TRIG;
	rtButtonManual						: R_TRIG;
	rtButtonMaintenance					: R_TRIG;
	rtButtonStart						: R_TRIG;
	rtButtonReset						: R_TRIG;
	rtButtonStop						: R_TRIG;

	// State change permissions
	bAllowChangeToManual				: BOOL;
	bAllowChangeToMaintenance			: BOOL;
	bAllowChangeToAutomatic				: BOOL;
	czas 								: ARRAY[0..100] OF TON;
	rtbAuto								: R_TRIG;
	bM_Start							: BOOL;
	seq									: INT;
END_VAR

// Triggers
rtButtonAutomatic(CLK:= bHMIModeRequest_Automatic );
rtButtonManual(CLK:= bHMIModeRequest_Manual );
rtButtonMaintenance(CLK:= bHMIModeRequest_Maintenance );
rtButtonStart(CLK:= bHMICommandRequest_Run);
rtButtonStop(CLK:= bHMICommandRequest_Stop);
rtButtonReset(CLK:= bHMICommandRequest_Reset);


//przepisanie zmiennych
bHMICommandRequest_Run:=GVL_IO.B1K1;
bHMICommandRequest_Stop:=GVL_IO.B1K3;
bHMICommandRequest_Reset :=GVL_IO.B1K8;
bHMIModeRequest_Automatic :=GVL_HMI.bAutoWybor;

// SAFETY niezaleznie
IF NOT GVL_SafetyFrom_RT2.bSAFETY_PermissionSS1 OR bHMICommandRequest_Abort THEN
	GVL_Machine.eCommand						:= E_MachineCommand.eAbort;
	GVL_Machine.eState							:= E_MachineState.eAborted;
END_IF

//uruchomienie automatu 

rtbAuto(CLK:=GVL_HMI.bAuto);
// przełączynik trybu auto/manual
IF GVL_HMI.bAuto THEN
	bHMIModeRequest_Automatic := TRUE;
	bHMIModeRequest_Manual := FALSE;
ELSE
	bHMIModeRequest_Automatic := FALSE;
	bHMIModeRequest_Manual := TRUE;
END_IF

CASE GVL_Machine.eMode OF 

	E_MachineMode.eAutomatic:

		// Zmiana trybu tylko gdy maszyna nie jest w Running
		IF GVL_Machine.eState <> E_MachineState.eRunning THEN
			IF rtButtonMaintenance.Q THEN
				GVL_Machine.eCommand			:= E_MachineCommand.eRestart;
				GVL_Machine.eMode				:= E_MachineMode.eMaintenance;
			END_IF
		END_IF
		
		IF GVL_Machine.eState <> E_MachineState.eRunning THEN
			IF rtButtonManual.Q THEN
				GVL_Machine.eCommand			:= E_MachineCommand.eRestart;
				GVL_Machine.eMode				:= E_MachineMode.eManual;
			END_IF
		END_IF
		//==============================================
		IF rtButtonStart.Q THEN 
			GVL_Machine.eCommand 	:= E_MachineCommand.eRun;
		END_IF

		IF rtButtonReset.Q AND GVL.bRestartRequired THEN
			GVL_Machine.eCommand	:= E_MachineCommand.eRestart;
		END_IF
		
		IF rtButtonReset.Q AND NOT GVL.bRestartRequired THEN
			GVL_Machine.eCommand	:= E_MachineCommand.eReset;
		END_IF
		
		IF GVL.bGeneralError OR GVL.bGeneralFatalError OR rtButtonStop.Q THEN
			GVL_Machine.eCommand	:= E_MachineCommand.eStop ;
		END_IF
		
	E_MachineMode.eMaintenance, E_MachineMode.eManual:
	
		// Reset, Restart, Error - not used
		
		// Zmiana trybu tylko gdy maszyna nie jest w Running
		IF GVL_Machine.eState <> E_MachineState.eRunning THEN
			IF rtButtonAutomatic.Q (* OR sth *) THEN
				GVL_Machine.eCommand			:= E_MachineCommand.eRestart;
				GVL_Machine.eMode				:= E_MachineMode.eAutomatic;
			END_IF
		END_IF
		
		//==============================================
		IF rtButtonStart.Q THEN 
			GVL_Machine.eCommand 	:= E_MachineCommand.eRun;
		END_IF

		IF rtButtonReset.Q AND GVL.bRestartRequired THEN
			GVL_Machine.eCommand	:= E_MachineCommand.eRestart;
		END_IF
		
		IF rtButtonReset.Q AND NOT GVL.bRestartRequired THEN
			GVL_Machine.eCommand	:= E_MachineCommand.eReset;
		END_IF
		
		IF rtButtonStop.Q THEN
			GVL_Machine.eCommand	:= E_MachineCommand.eStop ;
		END_IF

END_CASE

ACTION Act_CollectMachineState:
// Action to decide global machine state
GVL_Machine.eState; // :=
END_ACTION

ACTION Act_ModeChangeSelector:
bAllowChangeToManual 				:= NOT (P_Hbot_v3.eMachineState <> E_MachineState.eRunning); //
bAllowChangeToMaintenance;
bAllowChangeToAutomatic;
END_ACTION

END_PROGRAM

// ---- POUs/Programy/Hbot/P_Hbot_V3.TcPOU
PROGRAM P_Hbot_V3
VAR_INPUT
	eMachineMode							: E_MachineMode; 		// Machine mode
	eMachineCommand							: E_MachineCommand; 	// Command from top level state program
END_VAR
VAR_OUTPUT
	eMachineState							: E_MachineState;
  	bError									: BOOL;
END_VAR
VAR_IN_OUT

END_VAR
VAR
	// INPUTS
	bIn1									: BOOL;
	// OUTPUTS
	bOut1									: BOOL;	
	// Local
	iStateIdle								: INT;
	iStepStarting							: INT;
	iStateStoping							: INT;
	iStateAborting							: INT;	
// HMI Maintenance 
	
	// FBs Axis Online
	Axis_MCS_X						: AXIS_REF; 		// virtual axis X
	Axis_MCS_Y						: AXIS_REF;			// virtual axis Y
	Axis_ACS_X						: AXIS_REF;			// HW axis X
	Axis_ACS_Y						: AXIS_REF;			// HW axis Y
	stMcAxisOnline_MCS_X			: ST_McAxisOnline;
	stMcAxisOnline_MCS_Y			: ST_McAxisOnline;
	stMcAxisOnline_ACS_X			: ST_McAxisOnline;
	stMcAxisOnline_ACS_Y			: ST_McAxisOnline;
	


	fbMcAxisOnline_MCS_X			: FB_McAxisOnlineAX5000;
	fbMcAxisOnline_MCS_Y			: FB_McAxisOnlineAX5000;
	fbMcAxisOnline_ACS_X			: FB_McAxisOnlineAX5000;
	fbMcAxisOnline_ACS_Y			: FB_McAxisOnlineAX5000;

	tonAxesReady 					: TON;
	tonAxesError 					: TON;
	R_bReadyForMove					:R_Trig;


	
	rPickItemHigh			: REAL	:= GVL_Recipe.Poz_Z_Pobranie;
	rPlaceItemHigh			: REAL	:= GVL_Recipe.Poz_Z_Odlozenie;
	rItemPickVelocity		: REAL 	:= GVL_Recipe.Predk_plot_pobranie;//50
	rItemPlaceVelocity		: REAL 	:= GVL_Recipe.Predk_plot_odlozenie;//50
	rMoveVelocity			: REAL 	:= GVL_Recipe.Predk_plot_ruch;
	rMoveMode				: REAL 	:= 0;
	
	//Mode select
	bPickAndPlace			: BOOL;
	bReturnToPick			: BOOL;
	bReferneceHbot			: BOOL;
	
	//Status
	bReadyToPick			: BOOL;
	bReadyToPlace			: BOOL;
	bHome					: BOOL;
	bReadyForMove			: BOOL;
	bPicked					: BOOL;
	bPlaced					: BOOL;
	//CMDs
	bMoveCmd				: BOOL;
	bPickDone				: BOOL;
	bPlaceDone				: BOOL;
	bHomeDone				: BOOL;
	bPickedACK				: BOOL;
	bPlacedACK				: BOOL;
	bReadyToPickACK			: BOOL;
	bReadyToPlaceACK		: BOOL;
	
